# B&R Automation Studio project EFI (part 6)

### gAlrCore.mpalarmxcore - PC_any/mappServices/gAlrCore.mpalarmxcore
```
Element gAlrCore (Type=mpalarmxcore)
  mapp.AlarmX.Core.Configuration:
    [0]:
      Name = Dryer.Alarm.GenCritical
      Message = {$IAT/Dryer.Alarm.GenCritical}
      Code = 10001
      Severity = 1
      Behavior = PersistentAlarm
        Acknowledge = 0
        ReactionUntilAcknowledged = FALSE
        DataUpdate:
          Activation:
            TimeStamp = TRUE
            Snippets = TRUE
        Recording:
          ActiveToInactive = TRUE
          UnacknowledgedToAcknowledged = FALSE
          AcknowledgedToUnacknowledged = FALSE
    [1]:
      Name = Dryer.Alarm.GenStop
      Message = {$IAT/Dryer.Alarm.GenStop}
      Code = 10002
      Severity = 1
      Behavior = PersistentAlarm
        Acknowledge = 0
        ReactionUntilAcknowledged = FALSE
        DataUpdate:
          Activation:
            TimeStamp = TRUE
            Snippets = TRUE
        Recording:
          ActiveToInactive = TRUE
          UnacknowledgedToAcknowledged = FALSE
          AcknowledgedToUnacknowledged = FALSE
    [2]:
      Name = Dryer.Alarm.GenStopDrying
      Message = {$IAT/Dryer.Alarm.GenStopDrying}
      Code = 10003
      Severity = 1
      Behavior = PersistentAlarm
        Acknowledge = 0
        ReactionUntilAcknowledged = FALSE
        DataUpdate:
          Activation:
            TimeStamp = TRUE
            Snippets = TRUE
        Recording:
          ActiveToInactive = TRUE
          UnacknowledgedToAcknowledged = FALSE
          AcknowledgedToUnacknowledged = FALSE
    [3]:
      Name = Dryer.Alarm.FanBreakers
      Message = {$IAT/Dryer.Alarm.FanBreakers}
      Code = 10004
      Severity = 1
      Behavior = PersistentAlarm
        Acknowledge = 0
        ReactionUntilAcknowledged = FALSE
        DataUpdate:
          Activation:
            TimeStamp = TRUE
            Snippets = TRUE
        Recording:
          ActiveToInactive = TRUE
          UnacknowledgedToAcknowledged = FALSE
          AcknowledgedToUnacknowledged = FALSE
    [4]:
      Name = Dryer.Alarm.FansPsu
      Message = {$IAT/Dryer.Alarm.FansPsu}
      Code = 10005
      Severity = 1
      Behavior = PersistentAlarm
        Acknowledge = 0
        ReactionUntilAcknowledged = FALSE
        DataUpdate:
          Activation:
            TimeStamp = TRUE
            Snippets = TRUE
        Recording:
          ActiveToInactive = TRUE
          UnacknowledgedToAcknowledged = FALSE
          AcknowledgedToUnacknowledged = FALSE
    [5]:
      Name = Dryer.Alarm.MainPsu
      Message = {$IAT/Dryer.Alarm.MainPsu}
      Code = 10006
      Severity = 1
      Behavior = PersistentAlarm
        Acknowledge = 0
        ReactionUntilAcknowledged = FALSE
        DataUpdate:
          Activation:
            TimeStamp = TRUE
            Snippets = TRUE
        Recording:
          ActiveToInactive = TRUE
          UnacknowledgedToAcknowledged = FALSE
          AcknowledgedToUnacknowledged = FALSE
    [6]:
      Name = Dryer.Alarm.MountedMedia
      Message = {$IAT/Dryer.Alarm.MountedMedia}
      Code = 10007
      Severity = 1
      Behavior = PersistentAlarm
        Acknowledge = 0
        ReactionUntilAcknowledged = FALSE
        DataUpdate:
          Activation:
            TimeStamp = TRUE
            Snippets = TRUE
        Recording:
          ActiveToInactive = TRUE
          UnacknowledgedToAcknowledged = FALSE
          AcknowledgedToUnacknowledged = FALSE
    [7]:
      Name = Dryer.Alarm.EstopFront
      Message = {$IAT/Dryer.Alarm.EstopFront}
      Code = 10008
      Severity = 1
      Behavior = PersistentAlarm
        Acknowledge = 0
        ReactionUntilAcknowledged = FALSE
        DataUpdate:
          Activation:
            TimeStamp = TRUE
            Snippets = TRUE
        Recording:
          ActiveToInactive = TRUE
          UnacknowledgedToAcknowledged = FALSE
          AcknowledgedToUnacknowledged = FALSE
    [8]:
      Name = Dryer.Alarm.EstopRear
      Message = {$IAT/Dryer.Alarm.EstopRear}
      Code = 10009
      Severity = 1
      Behavior = PersistentAlarm
        Acknowledge = 0
        ReactionUntilAcknowledged = FALSE
        DataUpdate:
          Activation:
            TimeStamp = TRUE
            Snippets = TRUE
        Recording:
          ActiveToInactive = TRUE
          UnacknowledgedToAcknowledged = FALSE
          AcknowledgedToUnacknowledged = FALSE
    [9]:
      Name = Dryer.Alarm.EstopRemote
      Message = {$IAT/Dryer.Alarm.EstopRemote}
      Code = 10011
      Severity = 1
      Behavior = PersistentAlarm
        Acknowledge = 0
        ReactionUntilAcknowledged = FALSE
        DataUpdate:
          Activation:
            TimeStamp = TRUE
            Snippets = TRUE
        Recording:
          ActiveToInactive = TRUE
          UnacknowledgedToAcknowledged = FALSE
          AcknowledgedToUnacknowledged = FALSE
    [10]:
      Name = Dryer.Alarm.WrongPhysConfig
      Message = {$IAT/Dryer.Alarm.WrongPhysConfig}
      Code = 10012
      Severity = 1
      Behavior = PersistentAlarm
        Acknowledge = 0
        ReactionUntilAcknowledged = FALSE
        DataUpdate:
          Activation:
            TimeStamp = TRUE
            Snippets = TRUE
        Recording:
          ActiveToInactive = TRUE
          UnacknowledgedToAcknowledged = FALSE
          AcknowledgedToUnacknowledged = FALSE
    [11]:
      Name = Dryer.Alarm.OvertorqueBelt
      Message = {$IAT/Dryer.Alarm.OvertorqueBelt}
      Code = 10013
      Severity = 1
      Behavior = PersistentAlarm
        Acknowledge = 0
        ReactionUntilAcknowledged = FALSE
        DataUpdate:
          Activation:
            TimeStamp = TRUE
            Snippets = TRUE
        Recording:
          ActiveToInactive = TRUE
          UnacknowledgedToAcknowledged = FALSE
          AcknowledgedToUnacknowledged = FALSE
    [12]:
      Name = Dryer.Alarm.OverTempBeltFast
      Message = {$IAT/Dryer.Alarm.OverTempBeltFast}
      Code = 10014
      Severity = 1
      Behavior = PersistentAlarm
        Acknowledge = 0
        ReactionUntilAcknowledged = FALSE
        DataUpdate:
          Activation:
            TimeStamp = TRUE
            Snippets = TRUE
        Recording:
          ActiveToInactive = TRUE
          UnacknowledgedToAcknowledged = FALSE
          AcknowledgedToUnacknowledged = FALSE
    [13]:
      Name = Dryer.Alarm.OverTempBeltSlow
      Message = {$IAT/Dryer.Alarm.OverTempBeltSlow}
      Code = 10015
      Severity = 1
      Behavior = PersistentAlarm
        Acknowledge = 0
        ReactionUntilAcknowledged = FALSE
        DataUpdate:
          Activation:
            TimeStamp = TRUE
            Snippets = TRUE
        Recording:
          ActiveToInactive = TRUE
          UnacknowledgedToAcknowledged = FALSE
          AcknowledgedToUnacknowledged = FALSE
    [14]:
      Name = Dryer.Alarm.FansPsu80
      Message = {$IAT/Dryer.Alarm.FansPsu80}
      Code = 15001
      Severity = 2
      Behavior = PersistentAlarm
        Acknowledge = 0
        ReactionUntilAcknowledged = FALSE
        DataUpdate:
          Activation:
            TimeStamp = TRUE
            Snippets = TRUE
        Recording:
          ActiveToInactive = TRUE
          UnacknowledgedToAcknowledged = FALSE
          AcknowledgedToUnacknowledged = FALSE
    [15]:
      Name = Dryer.Warning.MountedMediaInside
      Message = {$IAT/Dryer.Warning.MountedMediaInside}
      Code = 15002
      Severity = 2
      Behavior = PersistentAlarm
        Acknowledge = 0
        ReactionUntilAcknowledged = FALSE
        DataUpdate:
          Activation:
            TimeStamp = TRUE
            Snippets = TRUE
        Recording:
          ActiveToInactive = TRUE
          UnacknowledgedToAcknowledged = FALSE
          AcknowledgedToUnacknowledged = FALSE
    [16]:
      Name = Dryer.Warning.BeltTempSensError
      Message = {$IAT/Dryer.Warning.BeltTempSensError}
      Code = 15003
      Severity = 2
      Behavior = PersistentAlarm
        Acknowledge = 0
        ReactionUntilAcknowledged = FALSE
        DataUpdate:
          Activation:
            TimeStamp = TRUE
            Snippets = TRUE
        Recording:
          ActiveToInactive = TRUE
          UnacknowledgedToAcknowledged = FALSE
          AcknowledgedToUnacknowledged = FALSE
    [17]:
      Name = Dryer.Warning.BoardInTempSensError
      Message = {$IAT/Dryer.Warning.BoardInTempSensError}
      Code = 15004
      Severity = 2
      Behavior = PersistentAlarm
        Acknowledge = 0
        ReactionUntilAcknowledged = FALSE
        DataUpdate:
          Activation:
            TimeStamp = TRUE
            Snippets = TRUE
        Recording:
          ActiveToInactive = TRUE
          UnacknowledgedToAcknowledged = FALSE
          AcknowledgedToUnacknowledged = FALSE
    [18]:
      Name = Dryer.Warning.BoardOutTempSensError
      Message = {$IAT/Dryer.Warning.BoardOutTempSensError}
      Code = 15005
      Severity = 2
      Behavior = PersistentAlarm
        Acknowledge = 0
        ReactionUntilAcknowledged = FALSE
        DataUpdate:
          Activation:
            TimeStamp = TRUE
            Snippets = TRUE
        Recording:
          ActiveToInactive = TRUE
          UnacknowledgedToAcknowledged = FALSE
          AcknowledgedToUnacknowledged = FALSE
    [19]:
      Name = Dryer.Warning.AirBlowerInTempSensError
      Message = {$IAT/Dryer.Warning.AirBlowerInTempSensError}
      Code = 15006
      Severity = 2
      Behavior = PersistentAlarm
        Acknowledge = 0
        ReactionUntilAcknowledged = FALSE
        DataUpdate:
          Activation:
            TimeStamp = TRUE
            Snippets = TRUE
        Recording:
          ActiveToInactive = TRUE
          UnacknowledgedToAcknowledged = FALSE
          AcknowledgedToUnacknowledged = FALSE
    [20]:
      Name = Dryer.Warning.AirBlowerOutTempSensError
      Message = {$IAT/Dryer.Warning.AirBlowerOutTempSensError}
      Code = 15007
      Severity = 2
      Behavior = PersistentAlarm
        Acknowledge = 0
        ReactionUntilAcknowledged = FALSE
        DataUpdate:
          Activation:
            TimeStamp = TRUE
            Snippets = TRUE
        Recording:
          ActiveToInactive = TRUE
          UnacknowledgedToAcknowledged = FALSE
          AcknowledgedToUnacknowledged = FALSE
    [21]:
      Name = Dryer.Warning.FrontDoorOpened
      Message = {$IAT/Dryer.Warning.FrontDoorOpened}
      Code = 15008
      Severity = 2
      Behavior = PersistentAlarm
        Acknowledge = 0
        ReactionUntilAcknowledged = FALSE
        DataUpdate:
          Activation:
            TimeStamp = TRUE
            Snippets = TRUE
        Recording:
          ActiveToInactive = TRUE
          UnacknowledgedToAcknowledged = FALSE
          AcknowledgedToUnacknowledged = FALSE
    [22]:
      Name = Dryer.Warning.RearDoorOpened
      Message = {$IAT/Dryer.Warning.RearDoorOpened}
      Code = 15009
      Severity = 2
      Behavior = PersistentAlarm
        Acknowledge = 0
        ReactionUntilAcknowledged = FALSE
        DataUpdate:
          Activation:
            TimeStamp = TRUE
            Snippets = TRUE
        Recording:
          ActiveToInactive = TRUE
          UnacknowledgedToAcknowledged = FALSE
          AcknowledgedToUnacknowledged = FALSE
    [23]:
      Name = Dryer.Warning.BentMedia
      Message = {$IAT/Dryer.Warning.BentMedia}
      Code = 15010
      Severity = 2
      Behavior = PersistentAlarm
        Acknowledge = 0
        ReactionUntilAcknowledged = FALSE
        DataUpdate:
          Activation:
            TimeStamp = TRUE
            Snippets = TRUE
        Recording:
          ActiveToInactive = TRUE
          UnacknowledgedToAcknowledged = FALSE
          AcknowledgedToUnacknowledged = FALSE
    [24]:
      Name = Dryer.Warning.NotMovementEnabled
      Message = {$IAT/Dryer.Warning.NotMovementEnabled}
      Code = 15011
      Severity = 2
      Behavior = PersistentAlarm
        Acknowledge = 0
        ReactionUntilAcknowledged = FALSE
        DataUpdate:
          Activation:
            TimeStamp = TRUE
            Snippets = TRUE
        Recording:
          ActiveToInactive = TRUE
          UnacknowledgedToAcknowledged = FALSE
          AcknowledgedToUnacknowledged = FALSE
    [25]:
      Name = Dryer.Warning.KeyMantenance
      Message = {$IAT/Dryer.Warning.KeyMantenance}
      Code = 15013
      Severity = 2
      Behavior = PersistentAlarm
        Acknowledge = 0
        ReactionUntilAcknowledged = FALSE
        DataUpdate:
          Activation:
            TimeStamp = TRUE
            Snippets = TRUE
        Recording:
          ActiveToInactive = TRUE
          UnacknowledgedToAcknowledged = FALSE
          AcknowledgedToUnacknowledged = FALSE
    [26]:
      Name = Dryer.Warning.JamLowCrash
      Message = {$IAT/Dryer.Warning.JamLowCrash}
      Code = 15014
      Severity = 2
      Behavior = PersistentAlarm
        Acknowledge = 0
        ReactionUntilAcknowledged = FALSE
        DataUpdate:
          Activation:
            TimeStamp = TRUE
            Snippets = TRUE
        Recording:
          ActiveToInactive = TRUE
          UnacknowledgedToAcknowledged = FALSE
          AcknowledgedToUnacknowledged = FALSE
    [27]:
      Name = Dryer.Alarm.BeltAnyDriveAlarm
      Message = {$IAT/Dryer.Alarm.BeltAnyDriveAlarm}
      Code = 30002
      Severity = 1
      Behavior = PersistentAlarm
        Acknowledge = 0
        ReactionUntilAcknowledged = FALSE
        DataUpdate:
          Activation:
            TimeStamp = TRUE
            Snippets = TRUE
        Recording:
          ActiveToInactive = TRUE
          UnacknowledgedToAcknowledged = FALSE
          AcknowledgedToUnacknowledged = FALSE
    [28]:
      Name = Dryer.Alarm.BeltAlrPowerBeltError
      Message = {$IAT/Dryer.Alarm.BeltAlrPowerBeltError}
      Code = 30003
      Severity = 1
      Behavior = PersistentAlarm
        Acknowledge = 0
        ReactionUntilAcknowledged = FALSE
        DataUpdate:
          Activation:
            TimeStamp = TRUE
            Snippets = TRUE
        Recording:
          ActiveToInactive = TRUE
          UnacknowledgedToAcknowledged = FALSE
          AcknowledgedToUnacknowledged = FALSE
    [29]:
      Name = Dryer.Alarm.BeltAlrComDrive
      Message = {$IAT/Dryer.Alarm.BeltAlrComDrive}
      Code = 30004
      Severity = 1
      Behavior = PersistentAlarm
        Acknowledge = 0
        ReactionUntilAcknowledged = FALSE
        DataUpdate:
          Activation:
            TimeStamp = TRUE
            Snippets = TRUE
        Recording:
          ActiveToInactive = TRUE
          UnacknowledgedToAcknowledged = FALSE
          AcknowledgedToUnacknowledged = FALSE
    [30]:
      Name = Dryer.Alarm.BeltAlrProtDrive
      Message = {$IAT/Dryer.Alarm.BeltAlrProtDrive}
      Code = 30005
      Severity = 1
      Behavior = PersistentAlarm
        Acknowledge = 0
        ReactionUntilAcknowledged = FALSE
        DataUpdate:
          Activation:
            TimeStamp = TRUE
            Snippets = TRUE
        Recording:
          ActiveToInactive = TRUE
          UnacknowledgedToAcknowledged = FALSE
          AcknowledgedToUnacknowledged = FALSE
    [31]:
      Name = Dryer.Alarm.BeltAlrOverTorque
      Message = {$IAT/Dryer.Alarm.BeltAlrOverTorque}
      Code = 30006
      Severity = 1
      Behavior = PersistentAlarm
        Acknowledge = 0
        ReactionUntilAcknowledged = FALSE
        DataUpdate:
          Activation:
            TimeStamp = TRUE
            Snippets = TRUE
        Recording:
          ActiveToInactive = TRUE
          UnacknowledgedToAcknowledged = FALSE
          AcknowledgedToUnacknowledged = FALSE
    [32]:
      Name = Dryer.Alarm.BeltBeltMotorTemp
      Message = {$IAT/Dryer.Alarm.BeltBeltMotorTemp}
      Code = 30007
      Severity = 1
      Behavior = PersistentAlarm
        Acknowledge = 0
        ReactionUntilAcknowledged = FALSE
        DataUpdate:
          Activation:
            TimeStamp = TRUE
            Snippets = TRUE
        Recording:
          ActiveToInactive = TRUE
          UnacknowledgedToAcknowledged = FALSE
          AcknowledgedToUnacknowledged = FALSE
    [33]:
      Name = Dryer.Alarm.BeltBeltDriverTemp
      Message = {$IAT/Dryer.Alarm.BeltBeltDriverTemp}
      Code = 30008
      Severity = 1
      Behavior = PersistentAlarm
        Acknowledge = 0
        ReactionUntilAcknowledged = FALSE
        DataUpdate:
          Activation:
            TimeStamp = TRUE
            Snippets = TRUE
        Recording:
          ActiveToInactive = TRUE
          UnacknowledgedToAcknowledged = FALSE
          AcknowledgedToUnacknowledged = FALSE
    [34]:
      Name = Dryer.Alarm.BeltNoPerimeter
      Message = {$IAT/Dryer.Alarm.BeltNoPerimeter}
      Code = 30009
      Severity = 2
      Behavior = PersistentAlarm
        Acknowledge = 0
        ReactionUntilAcknowledged = FALSE
        DataUpdate:
          Activation:
            TimeStamp = TRUE
            Snippets = TRUE
        Recording:
          ActiveToInactive = TRUE
          UnacknowledgedToAcknowledged = FALSE
          AcknowledgedToUnacknowledged = FALSE
    [35]:
      Name = Dryer.Alarm.BeltNoGearBox
      Message = {$IAT/Dryer.Alarm.BeltNoGearBox}
      Code = 30010
      Severity = 2
      Behavior = PersistentAlarm
        Acknowledge = 0
        ReactionUntilAcknowledged = FALSE
        DataUpdate:
          Activation:
            TimeStamp = TRUE
            Snippets = TRUE
        Recording:
          ActiveToInactive = TRUE
          UnacknowledgedToAcknowledged = FALSE
          AcknowledgedToUnacknowledged = FALSE
    [36]:
      Name = Dryer.Alarm.xWarningOvertoque
      Message = {$IAT/Dryer.Alarm.xWarningOvertoque}
      Code = 30102
      Severity = 2
      Behavior = PersistentAlarm
        Acknowledge = 0
        ReactionUntilAcknowledged = FALSE
        DataUpdate:
          Activation:
            TimeStamp = TRUE
            Snippets = TRUE
        Recording:
          ActiveToInactive = TRUE
          UnacknowledgedToAcknowledged = FALSE
          AcknowledgedToUnacknowledged = FALSE
    [37]:
      Name = Dryer.Alarm.SblockNotReferenced
      Message = {$IAT/Dryer.Alarm.SblockNotReferenced}
      Code = 40001
      Severity = 1
      Behavior = PersistentAlarm
        Acknowledge = 0
        ReactionUntilAcknowledged = FALSE
        DataUpdate:
          Activation:
            TimeStamp = TRUE
            Snippets = TRUE
        Recording:
          ActiveToInactive = TRUE
          UnacknowledgedToAcknowledged = FALSE
          AcknowledgedToUnacknowledged = FALSE
    [38]:
      Name = Dryer.Alarm.SblockNotCommsDrive
      Message = {$IAT/Dryer.Alarm.SblockNotCommsDrive}
      Code = 40002
      Severity = 1
      Behavior = PersistentAlarm
        Acknowledge = 0
        ReactionUntilAcknowledged = FALSE
        DataUpdate:
          Activation:
            TimeStamp = TRUE
            Snippets = TRUE
        Recording:
          ActiveToInactive = TRUE
          UnacknowledgedToAcknowledged = FALSE
          AcknowledgedToUnacknowledged = FALSE
    [39]:
      Name = Dryer.Alarm.SblockDriveBreaker
      Message = {$IAT/Dryer.Alarm.SblockDriveBreaker}
      Code = 40003
      Severity = 1
      Behavior = PersistentAlarm
        Acknowledge = 0
        ReactionUntilAcknowledged = FALSE
        DataUpdate:
          Activation:
            TimeStamp = TRUE
            Snippets = TRUE
        Recording:
          ActiveToInactive = TRUE
          UnacknowledgedToAcknowledged = FALSE
          AcknowledgedToUnacknowledged = FALSE
    [40]:
      Name = Dryer.Alarm.SblockHomeSensorError
      Message = {$IAT/Dryer.Alarm.SblockHomeSensorError}
      Code = 40004
      Severity = 1
      Behavior = PersistentAlarm
        Acknowledge = 0
        ReactionUntilAcknowledged = FALSE
        DataUpdate:
          Activation:
            TimeStamp = TRUE
            Snippets = TRUE
        Recording:
          ActiveToInactive = TRUE
          UnacknowledgedToAcknowledged = FALSE
          AcknowledgedToUnacknowledged = FALSE
    [41]:
      Name = Dryer.Alarm.SblockCheckHomeSensor
      Message = {$IAT/Dryer.Alarm.SblockCheckHomeSensor}
      Code = 40051
      Severity = 2
      Behavior = PersistentAlarm
        Acknowledge = 0
        ReactionUntilAcknowledged = FALSE
        DataUpdate:
          Activation:
            TimeStamp = TRUE
            Snippets = TRUE
        Recording:
          ActiveToInactive = TRUE
          UnacknowledgedToAcknowledged = FALSE
          AcknowledgedToUnacknowledged = FALSE
    [42]:
      Name = Dryer.Alarm.SblockMotorTemp
      Message = {$IAT/Dryer.Alarm.SblockMotorTemp}
      Code = 40052
      Severity = 2
      Behavior = PersistentAlarm
        Acknowledge = 0
        ReactionUntilAcknowledged = FALSE
        DataUpdate:
          Activation:
            TimeStamp = TRUE
            Snippets = TRUE
        Recording:
          ActiveToInactive = TRUE
          UnacknowledgedToAcknowledged = FALSE
          AcknowledgedToUnacknowledged = FALSE
    [43]:
      Name = Dryer.Alarm.SblockDriveTemp
      Message = {$IAT/Dryer.Alarm.SblockDriveTemp}
      Code = 40053
      Severity = 2
      Behavior = PersistentAlarm
        Acknowledge = 0
        ReactionUntilAcknowledged = FALSE
        DataUpdate:
          Activation:
            TimeStamp = TRUE
            Snippets = TRUE
        Recording:
          ActiveToInactive = TRUE
          UnacknowledgedToAcknowledged = FALSE
          AcknowledgedToUnacknowledged = FALSE
    [44]:
      Name = Dryer.Alarm.VaccSensor
      Message = {$IAT/Dryer.Alarm.VaccSensor}
      Code = 50001
      Severity = 1
      Behavior = PersistentAlarm
        Acknowledge = 0
        ReactionUntilAcknowledged = FALSE
        DataUpdate:
          Activation:
            TimeStamp = TRUE
            Snippets = TRUE
        Recording:
          ActiveToInactive = TRUE
          UnacknowledgedToAcknowledged = FALSE
          AcknowledgedToUnacknowledged = FALSE
    [45]:
      Name = Dryer.Alarm.VaccBlowerComsInput
      Message = {$IAT/Dryer.Alarm.VaccBlowerComsInput}
      Code = 50051
      Severity = 1
      Behavior = PersistentAlarm
        Acknowledge = 0
        ReactionUntilAcknowledged = FALSE
        DataUpdate:
          Activation:
            TimeStamp = TRUE
            Snippets = TRUE
        Recording:
          ActiveToInactive = TRUE
          UnacknowledgedToAcknowledged = FALSE
          AcknowledgedToUnacknowledged = FALSE
    [46]:
      Name = Dryer.Alarm.VaccBlowerComsOutput
      Message = {$IAT/Dryer.Alarm.VaccBlowerComsOutput}
      Code = 50052
      Severity = 1
      Behavior = PersistentAlarm
        Acknowledge = 0
        ReactionUntilAcknowledged = FALSE
        DataUpdate:
          Activation:
            TimeStamp = TRUE
            Snippets = TRUE
        Recording:
          ActiveToInactive = TRUE
          UnacknowledgedToAcknowledged = FALSE
          AcknowledgedToUnacknowledged = FALSE
    [47]:
      Name = Dryer.Alarm.VaccBlowerProtInput
      Message = {$IAT/Dryer.Alarm.VaccBlowerProtInput}
      Code = 50061
      Severity = 1
      Behavior = PersistentAlarm
        Acknowledge = 0
        ReactionUntilAcknowledged = FALSE
        DataUpdate:
          Activation:
            TimeStamp = TRUE
            Snippets = TRUE
        Recording:
          ActiveToInactive = TRUE
          UnacknowledgedToAcknowledged = FALSE
          AcknowledgedToUnacknowledged = FALSE
    [48]:
      Name = Dryer.Alarm.VaccBlowerProtOutput
      Message = {$IAT/Dryer.Alarm.VaccBlowerProtOutput}
      Code = 50062
      Severity = 1
      Behavior = PersistentAlarm
        Acknowledge = 0
        ReactionUntilAcknowledged = FALSE
        DataUpdate:
          Activation:
            TimeStamp = TRUE
            Snippets = TRUE
        Recording:
          ActiveToInactive = TRUE
          UnacknowledgedToAcknowledged = FALSE
          AcknowledgedToUnacknowledged = FALSE
    [49]:
      Name = Dryer.Alarm.VaccBlowerErrorInput
      Message = {$IAT/Dryer.Alarm.VaccBlowerErrorInput}
      Code = 50071
      Severity = 1
      Behavior = PersistentAlarm
        Acknowledge = 0
        ReactionUntilAcknowledged = FALSE
        DataUpdate:
          Activation:
            TimeStamp = TRUE
            Snippets = TRUE
        Recording:
          ActiveToInactive = TRUE
          UnacknowledgedToAcknowledged = FALSE
          AcknowledgedToUnacknowledged = FALSE
    [50]:
      Name = Dryer.Alarm.VaccBlowerErrorOutput
      Message = {$IAT/Dryer.Alarm.VaccBlowerErrorOutput}
      Code = 50072
      Severity = 1
      Behavior = PersistentAlarm
        Acknowledge = 0
        ReactionUntilAcknowledged = FALSE
        DataUpdate:
          Activation:
            TimeStamp = TRUE
            Snippets = TRUE
        Recording:
          ActiveToInactive = TRUE
          UnacknowledgedToAcknowledged = FALSE
          AcknowledgedToUnacknowledged = FALSE
    [51]:
      Name = Dryer.Alarm.VaccBlowerNotRunningInput
      Message = {$IAT/Dryer.Alarm.VaccBlowerNotRunningInput}
      Code = 50081
      Severity = 1
      Behavior = PersistentAlarm
        Acknowledge = 0
        ReactionUntilAcknowledged = FALSE
        DataUpdate:
          Activation:
            TimeStamp = TRUE
            Snippets = TRUE
        Recording:
          ActiveToInactive = TRUE
          UnacknowledgedToAcknowledged = FALSE
          AcknowledgedToUnacknowledged = FALSE
    [52]:
      Name = Dryer.Alarm.VaccBlowerNotRunningOutput
      Message = {$IAT/Dryer.Alarm.VaccBlowerNotRunningOutput}
      Code = 50082
      Severity = 1
      Behavior = PersistentAlarm
        Acknowledge = 0
        ReactionUntilAcknowledged = FALSE
        DataUpdate:
          Activation:
            TimeStamp = TRUE
            Snippets = TRUE
        Recording:
          ActiveToInactive = TRUE
          UnacknowledgedToAcknowledged = FALSE
          AcknowledgedToUnacknowledged = FALSE
    [53]:
      Name = Dryer.Alarm.NIRSafetyError
      Message = {$IAT/Dryer.Alarm.NIRSafetyError}
      Code = 60001
      Severity = 1
      Behavior = PersistentAlarm
        Acknowledge = 0
        ReactionUntilAcknowledged = FALSE
        DataUpdate:
          Activation:
            TimeStamp = TRUE
            Snippets = TRUE
        Recording:
          ActiveToInactive = TRUE
          UnacknowledgedToAcknowledged = FALSE
          AcknowledgedToUnacknowledged = FALSE
    [54]:
      Name = Dryer.Alarm.NIRFault
      Message = {$IAT/Dryer.Alarm.NIRFault}
      Code = 60002
      Severity = 1
      Behavior = PersistentAlarm
        Acknowledge = 0
        ReactionUntilAcknowledged = FALSE
        DataUpdate:
          Activation:
            TimeStamp = TRUE
            Snippets = TRUE
        Recording:
          ActiveToInactive = TRUE
          UnacknowledgedToAcknowledged = FALSE
          AcknowledgedToUnacknowledged = FALSE
    [55]:
      Name = Dryer.Alarm.NIRComsError
      Message = {$IAT/Dryer.Alarm.NIRComsError}
      Code = 60003
      Severity = 1
      Behavior = PersistentAlarm
        Acknowledge = 0
        ReactionUntilAcknowledged = FALSE
        DataUpdate:
          Activation:
            TimeStamp = TRUE
            Snippets = TRUE
        Recording:
          ActiveToInactive = TRUE
          UnacknowledgedToAcknowledged = FALSE
          AcknowledgedToUnacknowledged = FALSE
    [56]:
      Name = Dryer.Alarm.NIRInletHumiditySensError
      Message = {$IAT/Dryer.Alarm.NIRInletHumiditySensError}
      Code = 60021
      Severity = 2
      Behavior = PersistentAlarm
        Acknowledge = 0
        ReactionUntilAcknowledged = FALSE
        DataUpdate:
          Activation:
            TimeStamp = TRUE
            Snippets = TRUE
        Recording:
          ActiveToInactive = TRUE
          UnacknowledgedToAcknowledged = FALSE
          AcknowledgedToUnacknowledged = FALSE
    [57]:
      Name = Dryer.Alarm.NIRInletTempSensError
      Message = {$IAT/Dryer.Alarm.NIRInletTempSensError}
      Code = 60022
      Severity = 2
      Behavior = PersistentAlarm
        Acknowledge = 0
        ReactionUntilAcknowledged = FALSE
        DataUpdate:
          Activation:
            TimeStamp = TRUE
            Snippets = TRUE
        Recording:
          ActiveToInactive = TRUE
          UnacknowledgedToAcknowledged = FALSE
          AcknowledgedToUnacknowledged = FALSE
    [58]:
      Name = Dryer.Alarm.JamInputNIR1
      Message = {$IAT/Dryer.Alarm.JamInputNIR1}
      Code = 60051
      Severity = 1
      Behavior = PersistentAlarm
        Acknowledge = 0
        ReactionUntilAcknowledged = FALSE
        DataUpdate:
          Activation:
            TimeStamp = TRUE
            Snippets = TRUE
        Recording:
          ActiveToInactive = TRUE
          UnacknowledgedToAcknowledged = FALSE
          AcknowledgedToUnacknowledged = FALSE
    [59]:
      Name = Dryer.Alarm.JamOutputNIR1
      Message = {$IAT/Dryer.Alarm.JamOutputNIR1}
      Code = 60052
      Severity = 1
      Behavior = PersistentAlarm
        Acknowledge = 0
        ReactionUntilAcknowledged = FALSE
        DataUpdate:
          Activation:
            TimeStamp = TRUE
            Snippets = TRUE
        Recording:
          ActiveToInactive = TRUE
          UnacknowledgedToAcknowledged = FALSE
          AcknowledgedToUnacknowledged = FALSE
    [60]:
      Name = Dryer.Alarm.JamInputNIR2
      Message = {$IAT/Dryer.Alarm.JamInputNIR2}
      Code = 60061
      Severity = 1
      Behavior = PersistentAlarm
        Acknowledge = 0
        ReactionUntilAcknowledged = FALSE
        DataUpdate:
          Activation:
            TimeStamp = TRUE
            Snippets = TRUE
        Recording:
          ActiveToInactive = TRUE
          UnacknowledgedToAcknowledged = FALSE
          AcknowledgedToUnacknowledged = FALSE
    [61]:
      Name = Dryer.Alarm.JamOutputNIR2
      Message = {$IAT/Dryer.Alarm.JamOutputNIR2}
      Code = 60062
      Severity = 1
      Behavior = PersistentAlarm
        Acknowledge = 0
        ReactionUntilAcknowledged = FALSE
        DataUpdate:
          Activation:
            TimeStamp = TRUE
            Snippets = TRUE
        Recording:
          ActiveToInactive = TRUE
          UnacknowledgedToAcknowledged = FALSE
          AcknowledgedToUnacknowledged = FALSE
    [62]:
      Name = Dryer.Alarm.JamRearNIR1
      Message = {$IAT/Dryer.Alarm.JamRearNIR1}
      Code = 60071
      Severity = 1
      Behavior = PersistentAlarm
        Acknowledge = 0
        ReactionUntilAcknowledged = FALSE
        DataUpdate:
          Activation:
            TimeStamp = TRUE
            Snippets = TRUE
        Recording:
          ActiveToInactive = TRUE
          UnacknowledgedToAcknowledged = FALSE
          AcknowledgedToUnacknowledged = FALSE
    [63]:
      Name = Dryer.Alarm.JamRearNIR2
      Message = {$IAT/Dryer.Alarm.JamRearNIR2}
      Code = 60072
      Severity = 1
      Behavior = PersistentAlarm
        Acknowledge = 0
        ReactionUntilAcknowledged = FALSE
        DataUpdate:
          Activation:
            TimeStamp = TRUE
            Snippets = TRUE
        Recording:
          ActiveToInactive = TRUE
          UnacknowledgedToAcknowledged = FALSE
          AcknowledgedToUnacknowledged = FALSE
    [64]:
      Name = Dryer.Alarm.JamMechCrossNIR1
      Message = {$IAT/Dryer.Alarm.JamMechCrossNIR1}
      Code = 60081
      Severity = 1
      Behavior = PersistentAlarm
        Acknowledge = 0
        ReactionUntilAcknowledged = FALSE
        DataUpdate:
          Activation:
            TimeStamp = TRUE
            Snippets = TRUE
        Recording:
          ActiveToInactive = TRUE
          UnacknowledgedToAcknowledged = FALSE
          AcknowledgedToUnacknowledged = FALSE
    [65]:
      Name = Dryer.Alarm.JamMechCrossNIR2
      Message = {$IAT/Dryer.Alarm.JamMechCrossNIR2}
      Code = 60082
      Severity = 1
      Behavior = PersistentAlarm
        Acknowledge = 0
        ReactionUntilAcknowledged = FALSE
        DataUpdate:
          Activation:
            TimeStamp = TRUE
            Snippets = TRUE
        Recording:
          ActiveToInactive = TRUE
          UnacknowledgedToAcknowledged = FALSE
          AcknowledgedToUnacknowledged = FALSE
    [66]:
      Name = Dryer.Alarm.NIRSurfaceTemp1
      Message = {$IAT/Dryer.Alarm.NIRSurfaceTemp1}
      Code = 60101
      Severity = 2
      Behavior = PersistentAlarm
        Acknowledge = 0
        ReactionUntilAcknowledged = FALSE
        DataUpdate:
          Activation:
            TimeStamp = TRUE
            Snippets = TRUE
        Recording:
          ActiveToInactive = TRUE
          UnacknowledgedToAcknowledged = FALSE
          AcknowledgedToUnacknowledged = FALSE
    [67]:
      Name = Dryer.Alarm.NIRSurfaceTemp2
      Message = {$IAT/Dryer.Alarm.NIRSurfaceTemp2}
      Code = 60102
      Severity = 2
      Behavior = PersistentAlarm
        Acknowledge = 0
        ReactionUntilAcknowledged = FALSE
        DataUpdate:
          Activation:
            TimeStamp = TRUE
            Snippets = TRUE
        Recording:
          ActiveToInactive = TRUE
          UnacknowledgedToAcknowledged = FALSE
          AcknowledgedToUnacknowledged = FALSE
    [68]:
      Name = Dryer.Alarm.NIRSurfaceTempSensErr1
      Message = {$IAT/Dryer.Alarm.NIRSurfaceTempSensErr1}
      Code = 60111
      Severity = 2
      Behavior = PersistentAlarm
        Acknowledge = 0
        ReactionUntilAcknowledged = FALSE
        DataUpdate:
          Activation:
            TimeStamp = TRUE
            Snippets = TRUE
        Recording:
          ActiveToInactive = TRUE
          UnacknowledgedToAcknowledged = FALSE
          AcknowledgedToUnacknowledged = FALSE
    [69]:
      Name = Dryer.Alarm.NIRSurfaceTempSensErr2
      Message = {$IAT/Dryer.Alarm.NIRSurfaceTempSensErr2}
      Code = 60112
      Severity = 2
      Behavior = PersistentAlarm
        Acknowledge = 0
        ReactionUntilAcknowledged = FALSE
        DataUpdate:
          Activation:
            TimeStamp = TRUE
            Snippets = TRUE
        Recording:
          ActiveToInactive = TRUE
          UnacknowledgedToAcknowledged = FALSE
          AcknowledgedToUnacknowledged = FALSE
    [70]:
      Name = Dryer.Alarm.BlockedFan1Nir1
      Message = {$IAT/Dryer.Alarm.BlockedFan1Nir1}
      Code = 60201
      Severity = 2
      Behavior = PersistentAlarm
        Acknowledge = 0
        ReactionUntilAcknowledged = FALSE
        DataUpdate:
          Activation:
            TimeStamp = TRUE
            Snippets = TRUE
        Recording:
          ActiveToInactive = TRUE
          UnacknowledgedToAcknowledged = FALSE
          AcknowledgedToUnacknowledged = FALSE
    [71]:
      Name = Dryer.Alarm.BlockedFan2Nir1
      Message = {$IAT/Dryer.Alarm.BlockedFan2Nir1}
      Code = 60202
      Severity = 2
      Behavior = PersistentAlarm
        Acknowledge = 0
        ReactionUntilAcknowledged = FALSE
        DataUpdate:
          Activation:
            TimeStamp = TRUE
            Snippets = TRUE
        Recording:
          ActiveToInactive = TRUE
          UnacknowledgedToAcknowledged = FALSE
          AcknowledgedToUnacknowledged = FALSE
    [72]:
      Name = Dryer.Alarm.BlockedFan3Nir1
      Message = {$IAT/Dryer.Alarm.BlockedFan3Nir1}
      Code = 60203
      Severity = 2
      Behavior = PersistentAlarm
        Acknowledge = 0
        ReactionUntilAcknowledged = FALSE
        DataUpdate:
          Activation:
            TimeStamp = TRUE
            Snippets = TRUE
        Recording:
          ActiveToInactive = TRUE
          UnacknowledgedToAcknowledged = FALSE
          AcknowledgedToUnacknowledged = FALSE
    [73]:
      Name = Dryer.Alarm.BlockedFan4Nir1
      Message = {$IAT/Dryer.Alarm.BlockedFan4Nir1}
      Code = 60204
      Severity = 2
      Behavior = PersistentAlarm
        Acknowledge = 0
        ReactionUntilAcknowledged = FALSE
        DataUpdate:
          Activation:
            TimeStamp = TRUE
            Snippets = TRUE
        Recording:
          ActiveToInactive = TRUE
          UnacknowledgedToAcknowledged = FALSE
          AcknowledgedToUnacknowledged = FALSE
    [74]:
      Name = Dryer.Alarm.BlockedFan1Nir2
      Message = {$IAT/Dryer.Alarm.BlockedFan1Nir2}
      Code = 60211
      Severity = 2
      Behavior = PersistentAlarm
        Acknowledge = 0
        ReactionUntilAcknowledged = FALSE
        DataUpdate:
          Activation:
            TimeStamp = TRUE
            Snippets = TRUE
        Recording:
          ActiveToInactive = TRUE
          UnacknowledgedToAcknowledged = FALSE
          AcknowledgedToUnacknowledged = FALSE
    [75]:
      Name = Dryer.Alarm.BlockedFan2Nir2
      Message = {$IAT/Dryer.Alarm.BlockedFan2Nir2}
      Code = 60212
      Severity = 2
      Behavior = PersistentAlarm
        Acknowledge = 0
        ReactionUntilAcknowledged = FALSE
        DataUpdate:
          Activation:
            TimeStamp = TRUE
            Snippets = TRUE
        Recording:
          ActiveToInactive = TRUE
          UnacknowledgedToAcknowledged = FALSE
          AcknowledgedToUnacknowledged = FALSE
    [76]:
      Name = Dryer.Alarm.BlockedFan3Nir2
      Message = {$IAT/Dryer.Alarm.BlockedFan3Nir2}
      Code = 60213
      Severity = 2
      Behavior = PersistentAlarm
        Acknowledge = 0
        ReactionUntilAcknowledged = FALSE
        DataUpdate:
          Activation:
            TimeStamp = TRUE
            Snippets = TRUE
        Recording:
          ActiveToInactive = TRUE
          UnacknowledgedToAcknowledged = FALSE
          AcknowledgedToUnacknowledged = FALSE
    [77]:
      Name = Dryer.Alarm.BlockedFan4Nir2
      Message = {$IAT/Dryer.Alarm.BlockedFan4Nir2}
      Code = 60214
      Severity = 2
      Behavior = PersistentAlarm
        Acknowledge = 0
        ReactionUntilAcknowledged = FALSE
        DataUpdate:
          Activation:
            TimeStamp = TRUE
            Snippets = TRUE
        Recording:
          ActiveToInactive = TRUE
          UnacknowledgedToAcknowledged = FALSE
          AcknowledgedToUnacknowledged = FALSE
    [78]:
      Name = Dryer.Alarm.ArcLampComsError
      Message = {$IAT/Dryer.Alarm.ArcLampComsError}
      Code = 70001
      Severity = 1
      Behavior = PersistentAlarm
        Acknowledge = 0
        ReactionUntilAcknowledged = FALSE
        DataUpdate:
          Activation:
            TimeStamp = TRUE
            Snippets = TRUE
        Recording:
          ActiveToInactive = TRUE
          UnacknowledgedToAcknowledged = FALSE
          AcknowledgedToUnacknowledged = FALSE
    [79]:
      Name = Dryer.Alarm.ArcLampCredentialsError
      Message = {$IAT/Dryer.Alarm.ArcLampCredentialsError}
      Code = 70002
      Severity = 1
      Behavior = PersistentAlarm
        Acknowledge = 0
        ReactionUntilAcknowledged = FALSE
        DataUpdate:
          Activation:
            TimeStamp = TRUE
            Snippets = TRUE
        Recording:
          ActiveToInactive = TRUE
          UnacknowledgedToAcknowledged = FALSE
          AcknowledgedToUnacknowledged = FALSE
    [80]:
      Name = Dryer.Alarm.ArcLampInternalError
      Message = {$IAT/Dryer.Alarm.ArcLampInternalError}
      Code = 70003
      Severity = 1
      Behavior = PersistentAlarm
        Acknowledge = 0
        ReactionUntilAcknowledged = FALSE
        DataUpdate:
          Activation:
            TimeStamp = TRUE
            Snippets = TRUE
        Recording:
          ActiveToInactive = TRUE
          UnacknowledgedToAcknowledged = FALSE
          AcknowledgedToUnacknowledged = FALSE
    [81]:
      Name = Dryer.Alarm.ArcLampJam
      Message = {$IAT/Dryer.Alarm.ArcLampJam}
      Code = 70004
      Severity = 1
      Behavior = PersistentAlarm
        Acknowledge = 0
        ReactionUntilAcknowledged = FALSE
        DataUpdate:
          Activation:
            TimeStamp = TRUE
            Snippets = TRUE
        Recording:
          ActiveToInactive = TRUE
          UnacknowledgedToAcknowledged = FALSE
          AcknowledgedToUnacknowledged = FALSE
    [82]:
      Name = Dryer.Alarm.ArcLampAlarmLamp1
      Message = {$IAT/Dryer.Alarm.ArcLampAlarmLamp1}
      Code = 70051
      Severity = 1
      Behavior = PersistentAlarm
        Acknowledge = 0
        ReactionUntilAcknowledged = FALSE
        DataUpdate:
          Activation:
            TimeStamp = TRUE
            Snippets = TRUE
        Recording:
          ActiveToInactive = TRUE
          UnacknowledgedToAcknowledged = FALSE
          AcknowledgedToUnacknowledged = FALSE
    [83]:
      Name = Dryer.Alarm.ArcLampAlarmLamp2
      Message = {$IAT/Dryer.Alarm.ArcLampAlarmLamp2}
      Code = 70052
      Severity = 1
      Behavior = PersistentAlarm
        Acknowledge = 0
        ReactionUntilAcknowledged = FALSE
        DataUpdate:
          Activation:
            TimeStamp = TRUE
            Snippets = TRUE
        Recording:
          ActiveToInactive = TRUE
          UnacknowledgedToAcknowledged = FALSE
          AcknowledgedToUnacknowledged = FALSE
    [84]:
      Name = Dryer.Alarm.CheckMediaExit1
      Message = {$IAT/Dryer.Alarm.CheckMediaExit1}
      Code = 80001
      Severity = 1
      Behavior = PersistentAlarm
        Acknowledge = 0
        ReactionUntilAcknowledged = FALSE
        DataUpdate:
          Activation:
            TimeStamp = TRUE
            Snippets = TRUE
        Recording:
          ActiveToInactive = TRUE
          UnacknowledgedToAcknowledged = FALSE
          AcknowledgedToUnacknowledged = FALSE
    [85]:
      Name = Dryer.Alarm.CheckMediaExit2
      Message = {$IAT/Dryer.Alarm.CheckMediaExit2}
      Code = 80002
      Severity = 1
      Behavior = PersistentAlarm
        Acknowledge = 0
        ReactionUntilAcknowledged = FALSE
        DataUpdate:
          Activation:
            TimeStamp = TRUE
            Snippets = TRUE
        Recording:
          ActiveToInactive = TRUE
          UnacknowledgedToAcknowledged = FALSE
          AcknowledgedToUnacknowledged = FALSE
  mapp.AlarmX.Core.Categories:
    [0]:
      Name = Critical
      SourceProperty:
        Severity = 1
    [1]:
      Name = Warning
      SourceProperty:
        Severity = 2
    [2]:
      Name = Message
      SourceProperty:
        Severity = 3
```

### gAlrHist.mpalarmxhistory - PC_any/mappServices/gAlrHist.mpalarmxhistory
```
Element gAlrHist (Type=mpalarmxhistory)
  mapp.AlarmX.History:
    Memory:
      MemorySize = 600
```

## Configuration SimTests

CPU , AutomationRuntime K4.93, Build 4.1.2, Safety 0.0, Vc V4.73.2

### Task classes (Cpu.sw)
```
Cyclic#1 (cycle 4000 us, tolerance 0 us):
  mappHMI <- (binary)
Cyclic#2 (cycle 8000 us, tolerance 0 us):
  Initialize <- Printer.Config.Initialize.prg
  InitAxisCo <- ExtPack._Motion.AxisCtrl.AxisCtrl_v2.InitAxisControl.prg
  Belt <- ExtPack._Motion.AxisCtrl.AxisCtrl_v2.AxisCtrl.prg
  BK_A <- ExtPack._Motion.AxisCtrl.AxisCtrl_v2.AxisCtrl.prg
  BK_B <- ExtPack._Motion.AxisCtrl.AxisCtrl_v2.AxisCtrl.prg
  Stepper3L <- ExtPack._Motion.AxisCtrl.AxisCtrl_v2.AxisCtrl.prg
  Gear3L <- ExtPack._Motion.AxisCtrl.AxisCtrl_v2.AxisCtrl.prg
  NoCrash1 <- ExtPack._Motion.AxisCtrl.AxisCtrl_v2.AxisCtrl.prg
  NoCrash2 <- ExtPack._Motion.AxisCtrl.AxisCtrl_v2.AxisCtrl.prg
  InitInvert <- ExtPack._Motion.InverterCtrl.InverterCtrl_v1.InitInverterCtrl.prg
  Inverter1 <- ExtPack._Motion.InverterCtrl.InverterCtrl_v1.InverterCtrl.prg
  Inverter2 <- ExtPack._Motion.InverterCtrl.InverterCtrl_v1.InverterCtrl.prg
  Inverter3 <- ExtPack._Motion.InverterCtrl.InverterCtrl_v1.InverterCtrl.prg
  Inverter4 <- ExtPack._Motion.InverterCtrl.InverterCtrl_v1.InverterCtrl.prg
  InitIclaSi <- ExtPack._Motion.IclaCtrl.IclaSim.IclaSim_v1.InitIclaSim.prg
  IclaSim1 <- ExtPack._Motion.IclaCtrl.IclaSim.IclaSim_v1.IclaSim.prg
  IclaSim2 <- ExtPack._Motion.IclaCtrl.IclaSim.IclaSim_v1.IclaSim.prg
  IclanLas <- ExtPack._Motion.IclaCtrl.IclaSim.IclaSim_v1.IclaSim.prg
  IclaEhd1 <- ExtPack._Motion.IclaCtrl.IclaSim.IclaSim_v1.IclaSim.prg
  IclaEhd2 <- ExtPack._Motion.IclaCtrl.IclaSim.IclaSim_v1.IclaSim.prg
  IclaEhd3 <- ExtPack._Motion.IclaCtrl.IclaSim.IclaSim_v1.IclaSim.prg
  IclaEhd4 <- ExtPack._Motion.IclaCtrl.IclaSim.IclaSim_v1.IclaSim.prg
  SimMachFst <- Printer.Sim.SimMachine_Fast.prg
  Analog_Fas <- ExtPack._Media.AnalogThicknessCtrl.AnalogThicknessCtrl_v1.Analog_Fast.prg
  nSens_Fast <- ExtPack._Media.nSensorCtrl.nSensorCtrl_v2.nSensorCtrl_Fast.prg
  Thick_Fast <- ExtPack._Media.ThicknessCtrl.ThicknessCtrl_v2.ThicknessCtrl_Fast.prg
Cyclic#4 (cycle 32000 us, tolerance 32000 us):
  PhysInp <- Printer.PhysicalMapping.PhysicalMapInputs.prg
  BlockInp <- Printer.BlockSignalsManager.BlockInputsMapping.prg
  SimMachine <- Printer.Sim.SimMachine.prg
  ThickSim <- ExtPack._Media.ThicknessCtrl.ThicknessCtrlSim.ThicknessCtrlSim_v1.ThicknessCtrlSim.prg
  ThickPos <- ExtPack._Media.ThicknessCtrl.ThicknessCtrl_v2.ThicknessCtrl.prg  // Thickness array manager
  LineCtrl <- LineCtrl.LineCtrl.prg
  Mach_Fast <- Printer.MachineCtrl.MachineCtrl_Fast.prg
  BeltCtrl <- ExtPack._Transport.BeltCtrl.BeltCtrl_v1.BeltCtrl.prg
  InitBlockC <- ExtPack.BlockCtrl.BlockCtrl_v1.InitBlockCtrl.prg
  Block_BK1 <- ExtPack.BlockCtrl.BlockCtrl_v1.BlockCtrl.prg
  Block_BK2 <- ExtPack.BlockCtrl.BlockCtrl_v1.BlockCtrl.prg
  AnalogThic <- ExtPack._Media.AnalogThicknessCtrl.AnalogThicknessCtrl_v1.AnalogThickness.prg
  nSensorCtr <- ExtPack._Media.nSensorCtrl.nSensorCtrl_v2.nSensorCtrl.prg
  InitChille <- ExtPack._Extras.ChillerCtrl.ChillerCtrl_v2.InitChiller.prg
  Chiller1 <- ExtPack._Extras.ChillerCtrl.ChillerCtrl_v2.ChillerCtrl.prg
  Chiller2 <- ExtPack._Extras.ChillerCtrl.ChillerCtrl_v2.ChillerCtrl.prg
  InitTransV <- ExtPack._Transport.TransVacuumCtrl.TransVacuumCtrl_v1.InitTransVacuumCtrl.prg
  TransVac1 <- ExtPack._Transport.TransVacuumCtrl.TransVacuumCtrl_v1.TransVacuumCtrl.prg
  TransVac2 <- ExtPack._Transport.TransVacuumCtrl.TransVacuumCtrl_v1.TransVacuumCtrl.prg
  InitNCrash <- ExtPack._Transport.NonCrashCtrl.NonCrashCtrl_v1.InitNonCrashCtrl.prg
  NonCrash1 <- ExtPack._Transport.NonCrashCtrl.NonCrashCtrl_v1.NonCrashCtrl.prg
  InitCuring <- ExtPack._Cure.CuringLedCtrl.CuringLedCtrl_v1.InitCuringLedCtrl.prg
  CuringLed1 <- ExtPack._Cure.CuringLedCtrl.CuringLedCtrl_v1.CuringLedCtrl.prg
  CuringLed2 <- ExtPack._Cure.CuringLedCtrl.CuringLedCtrl_v1.CuringLedCtrl.prg
  CuringLed3 <- ExtPack._Cure.CuringLedCtrl.CuringLedCtrl_v1.CuringLedCtrl.prg
  BlockOut <- Printer.BlockSignalsManager.BlockOutputsMapping.prg
  PhysOut <- Printer.PhysicalMapping.PhysicalMapOutputs.prg
  InitTraySi <- ExtPack._Tools.TestBench.TraySim.TraySim_v1.InitTraySim.prg
  TraySim1 <- ExtPack._Tools.TestBench.TraySim.TraySim_v1.TraySim.prg
  TraySim2 <- ExtPack._Tools.TestBench.TraySim.TraySim_v1.TraySim.prg
  InitBlockS <- ExtPack.BlockCtrl.BlockSim.BlockSim_v1.InitBlockSim.prg
  BlockSim1 <- ExtPack.BlockCtrl.BlockSim.BlockSim_v1.BlockSim.prg
  BlockSim2 <- ExtPack.BlockCtrl.BlockSim.BlockSim_v1.BlockSim.prg
  EhdCtrl <- ExtPack._Transport.EdgeHoldDown.EdgeHoldDown_v1.EdgeHoldDown.prg
  InitPaired <- ExtPack._Transport.PairedIclaMotors.PairedIclaMotors_v1.InitPairedIclaMotors.prg
  PairedIcl1 <- ExtPack._Transport.PairedIclaMotors.PairedIclaMotors_v1.PairedIclaMotors.prg
  PairedIcl2 <- ExtPack._Transport.PairedIclaMotors.PairedIclaMotors_v1.PairedIclaMotors.prg
  InitChilSi <- ExtPack._Extras.ChillerCtrl.ChillerSim.ChillerSim_v1.InitChillerSim.prg
  ChillSim1 <- ExtPack._Extras.ChillerCtrl.ChillerSim.ChillerSim_v1.ChillerSim.prg
  ChillSim2 <- ExtPack._Extras.ChillerCtrl.ChillerSim.ChillerSim_v1.ChillerSim.prg
  InitTrSim <- ExtPack._Transport.TransVacuumCtrl.TransVacuumSim.TransVacuumSim_v1.InitTransVacuumSim.prg
  TrVacSim1 <- ExtPack._Transport.TransVacuumCtrl.TransVacuumSim.TransVacuumSim_v1.TransVacuumSim.prg
  TrVacSim2 <- ExtPack._Transport.TransVacuumCtrl.TransVacuumSim.TransVacuumSim_v1.TransVacuumSim.prg
  TrVacSim3 <- ExtPack._Transport.TransVacuumCtrl.TransVacuumSim.TransVacuumSim_v1.TransVacuumSim.prg
  TrVacSim4 <- ExtPack._Transport.TransVacuumCtrl.TransVacuumSim.TransVacuumSim_v1.TransVacuumSim.prg
  InitCurSim <- ExtPack._Cure.CuringLedCtrl.CuringLedSim.CuringLedSim_v1.InitCuringLedSim.prg
  CurinSim1 <- ExtPack._Cure.CuringLedCtrl.CuringLedSim.CuringLedSim_v1.CuringLedSim.prg
  CurinSim2 <- ExtPack._Cure.CuringLedCtrl.CuringLedSim.CuringLedSim_v1.CuringLedSim.prg
  CurinSim3 <- ExtPack._Cure.CuringLedCtrl.CuringLedSim.CuringLedSim_v1.CuringLedSim.prg
  FeederCtrl <- ExtPack._Ancillaries.FeederCtrl.FeederCtrl_v1.FeederCtrl.prg
  PrimerCtrl <- ExtPack._Ancillaries.PrimerCtrl.PrimerCtrl_v1.PrimerCtrl.prg
  SarmCtrl <- ExtPack._Ancillaries.SarmCtrl.SarmCtrl.SarmCtrl.prg
  OpvCtrl <- ExtPack._Ancillaries.OpvCtrl.OpvCtrl_v1.OpvCtrl.prg
  StackerCtr <- ExtPack._Ancillaries.StackerCtrl.StackerCtrl_v1.StackerCtrl.prg
  DryerCtrl <- ExtPack._Ancillaries.DryerCtrl.DryerCtrl_v1.DryerCtrl.prg
  FeederSim <- ExtPack._Ancillaries.FeederCtrl.FeederSim.FeederSim_v1.FeederSim.prg
  SarmSim <- ExtPack._Ancillaries.SarmCtrl.SarmSim.SarmSim_v1.SarmSim.prg
  DryerSim <- Dryer.DryerSimAnc.DryerSimAnc_v1.DryerSimAnc.prg
  PrimerSim <- ExtPack._Ancillaries.PrimerCtrl.PrimerSim.PrimerSim_v1.PrimerSim.prg
  OpvSim <- ExtPack._Ancillaries.OpvCtrl.OpvSim.OpvSim_v1.OpvSim.prg
  SafeCtlSim <- ExtPack._Extras.SafetyControllerCtrl.SafetyControllerSim.SafetyControllerSim_v1.SafetyControllerSim.prg
  StackerSim <- ExtPack._Ancillaries.StackerCtrl.StackerSim.StackerSim_v1.StackerSim.prg
  InitJamDet <- ExtPack._Transport.JamDetectCtrl.JamDetect_v1.InitJamDetect.prg
  JamDetect1 <- ExtPack._Transport.JamDetectCtrl.JamDetect_v1.JamDetect.prg
  JamDetect2 <- ExtPack._Transport.JamDetectCtrl.JamDetect_v1.JamDetect.prg
  JamDetect3 <- ExtPack._Transport.JamDetectCtrl.JamDetect_v1.JamDetect.prg
  JamDetect4 <- ExtPack._Transport.JamDetectCtrl.JamDetect_v1.JamDetect.prg
  InitJamDeS <- ExtPack._Transport.JamDetectCtrl.JamDetectSim.JamDetectSim_v1.InitJamDetectSim.prg
  JamDetctS1 <- ExtPack._Transport.JamDetectCtrl.JamDetectSim.JamDetectSim_v1.JamDetectSim.prg
  JamDetctS2 <- ExtPack._Transport.JamDetectCtrl.JamDetectSim.JamDetectSim_v1.JamDetectSim.prg
  JamDetctS3 <- ExtPack._Transport.JamDetectCtrl.JamDetectSim.JamDetectSim_v1.JamDetectSim.prg
  JamDetctS4 <- ExtPack._Transport.JamDetectCtrl.JamDetectSim.JamDetectSim_v1.JamDetectSim.prg
  nSensorSim <- ExtPack._Media.nSensorCtrl.nSensorSim.nSensorSim_v1.nSensorSim.prg
  EhdSim <- ExtPack._Transport.EdgeHoldDown.EdgeHoldDownSim.EdgeHoldDownSim_v1.EdgeHoldDownSim.prg
  IniPairSim <- ExtPack._Transport.PairedIclaMotors.PairedIclaMotorsSim.PairedIclaMotorsSim_v1.InitPairedIclaMotorsSim.prg
  PairSim <- ExtPack._Transport.PairedIclaMotors.PairedIclaMotorsSim.PairedIclaMotorsSim_v1.PairedIclaMotorsSim.prg
  PairSim2 <- ExtPack._Transport.PairedIclaMotors.PairedIclaMotorsSim.PairedIclaMotorsSim_v1.PairedIclaMotorsSim.prg
  InitNonCra <- ExtPack._Transport.NonCrashCtrl.NonCrashSim.NonCrashSim_v1.InitNonCrashSim.prg
  NonCrashS1 <- ExtPack._Transport.NonCrashCtrl.NonCrashSim.NonCrashSim_v1.NonCrashSim.prg
Cyclic#5 (cycle 80000 us, tolerance 80000 us):
  InksInputs <- Printer.InksSignals.InksInputs.prg
  InitInksSi <- ExtPack.InksCtrl.InksSim.InksSim_v1.InitInksSim.prg
  InksSim01 <- ExtPack.InksCtrl.InksSim.InksSim_v1.InksSim.prg
  InksSim02 <- ExtPack.InksCtrl.InksSim.InksSim_v1.InksSim.prg
  InksSim03 <- ExtPack.InksCtrl.InksSim.InksSim_v1.InksSim.prg
  InksSim04 <- ExtPack.InksCtrl.InksSim.InksSim_v1.InksSim.prg
  InksSim05 <- ExtPack.InksCtrl.InksSim.InksSim_v1.InksSim.prg
  InksSim06 <- ExtPack.InksCtrl.InksSim.InksSim_v1.InksSim.prg
  InksSim07 <- ExtPack.InksCtrl.InksSim.InksSim_v1.InksSim.prg
  InksSim08 <- ExtPack.InksCtrl.InksSim.InksSim_v1.InksSim.prg
  InitIndex <- ExtPack.InksCtrl.InksCtrl_v3.InitInksCtrl.prg
  Inks_01 <- ExtPack.InksCtrl.InksCtrl_v3.InksCtrl.prg
  Inks_02 <- ExtPack.InksCtrl.InksCtrl_v3.InksCtrl.prg
  Inks_03 <- ExtPack.InksCtrl.InksCtrl_v3.InksCtrl.prg
  Inks_04 <- ExtPack.InksCtrl.InksCtrl_v3.InksCtrl.prg
  Inks_05 <- ExtPack.InksCtrl.InksCtrl_v3.InksCtrl.prg
  Inks_06 <- ExtPack.InksCtrl.InksCtrl_v3.InksCtrl.prg
  Inks_07 <- ExtPack.InksCtrl.InksCtrl_v3.InksCtrl.prg
  Inks_08 <- ExtPack.InksCtrl.InksCtrl_v3.InksCtrl.prg
  InksOutput <- Printer.InksSignals.InksOutputs.prg  // Physical outputs inks
  SafetySamp <- AsSafetySolution.SafetySample.prg
  EventLogGe <- ExtPack._Tools.EventLog.EventLog_v1.EventLogGen.prg
  SavePerman <- Printer.Config.SavePermanent.prg
  SimUseReg <- ExtPack._Tools.SimUseRegister.SimUseRegister_1.SimUseRegister.prg
Cyclic#6 (cycle 88000 us, tolerance 88000 us):
  SafetyCont <- ExtPack._Extras.SafetyControllerCtrl.SafetyControllerCtrl_v1.SafetyControllerCtrl.prg
  InitPowerM <- ExtPack._Extras.PowerMeterCtrl.PowerMeterCtrl_v1.InitPowerMeterCtrl.prg
  PowerMete1 <- ExtPack._Extras.PowerMeterCtrl.PowerMeterCtrl_v1.PowerMeterCtrl.prg
  PowerMete2 <- ExtPack._Extras.PowerMeterCtrl.PowerMeterCtrl_v1.PowerMeterCtrl.prg
  Mach_Conf <- Printer.Config.MachineConfigurator.prg  // Printer configurator program
  Mach_Slow <- Printer.MachineCtrl.MachineCtrl_Slow.prg
  ThickReadE <- ExtPack._Media.ThicknessCtrl.ThicknessCtrl_v2.ThickReadEnergy.prg
  BeltClean <- ExtPack._Transport.BeltCleaning.BeltCleaning_v1.BeltCleaning.prg
  BCleanSim <- ExtPack._Transport.BeltCleaning.BeltCleaningSim.BeltCleaningSim.prg
Cyclic#7 (cycle 44000 us, tolerance 88000 us):
  PLC2Kernel <- Printer.Comms.PLC2Kernel.prg
  ServModbus <- ExtPack._Comms.ModbusComms.ModbusComms_v1.ServModbus.prg
  Kernel2PLC <- Printer.Comms.Kernel2PLC.prg  // Comns Kernel to PLC
Cyclic#8 (cycle 16000 us, tolerance 16000 us):
  FunctionsT <- UnitTest.Tests.FunctionsTests.prg
  PrePrepare <- UnitTest.Tests.PrePrepare.prg
  PrepMach <- UnitTest.Tests.PrepareMachine.prg  // Prepare Machine to work properly in Sim
  BeltTests <- UnitTest.Tests.BeltTests.prg
  ConsTests <- UnitTest.Tests.ConsentTests.prg
  CleaningTe <- UnitTest.Tests.CleaningTests.prg
  LineTests <- UnitTest.Tests.LineTests.prg
  TrVacuumTe <- UnitTest.Tests.TrVacuumTests.prg
  BlockTests <- UnitTest.Tests.BlockTests.prg
  Cube <- UnitTest.Tests.Cube.prg
DataObjects: Acp10sys
NcDataObjects: AcpErrTxt <- AxisTables.AcpErrTxt.dob, acp10etxen <- AxisTables.acp10etxen.dob, SM_a <- AxisTables.SM_a.dob, SM_i <- AxisTables.SM_i.dob, BeltP4_a <- AxisTables.BeltP4_a.dob, BeltP4_i <- AxisTables.BeltP4_i.dob, BK1_a <- AxisTables.BK1_a.dob, BK1_i <- AxisTables.BK1_i.dob, BK_sim_a <- AxisTables.BK_sim_a.dob, NonCrash_a <- AxisTables.NonCrash_a.dob, NonCrash_i <- AxisTables.NonCrash_i.dob
VcDataObjects: SimVis <- Printer.Sim.SimVisu.dob, Panel <- AsSafetySolution.Panel.dob
Binaries: TCData, udbdef, vcfntttf, vcfile, vcshared, vcpdvnc, vcgclass, arial, SimVis03, arialxsr, vccslider, vcdsint, SimVis01, vccbtn, vcdsloc, vcpfar00, vccovl, vcmgr, vcctext, vcalarm, vcbclass, vcrt, vccnum, arialbd, vccshape, vcpdsw, vcnet, SimVis02, vctcal, vcpkat, vccstr, vcclbox, vccdt, vccurl, vccline, vccbar, vcchtml, vcxml, vccalarm, vcctrend, vccbmp, vccgauge, Panel01, Panel03, Panel02, vccddbox, vccpopup, TCLang, mvLoader, OpcUaSrv, arsvcreg, Acp10map, acp10cfg, User, Role, TC, ashwac, sysconf, ashwd, arconfig, asfw, iomap, Visu02, Visu03, Visu01, Diagn02, Diagn03, Diagn01, vcchspot, OpcUaMap
Libraries: UnitTest, LibAssert1, EFIAssert, UtWs, UtMgr, AsCANopen, FBs, Functions, ConvertFun, runtime, brsystem, sys_lib, standard, AsSafety, FileIO, AsXml, astime, asstring, AsFifo, NcGlobal, AsBrStr, BRSE_MBT, BRSE_MB, MTBasics, MTTypes, MTFilter, AsIecCon, AsIOAcc, AsBrMath, AsEPL, ArEventLog, Acp10_MC, Acp10par, Acp10sim, Acp10sdc, DataObj, EvLogLib, ArProject, AxisFunc, dvframe, AsSem, IecCheck, ThickLib, ErrACS380, Acp10man, MpAlarmX, MpBase, MpCom, MpServer, powerlnk, arssl, vcresman, ashttp, astcp, asopcuac, asopcuas, asmath, aruser, ashw, asarcfg
```

### Hardware
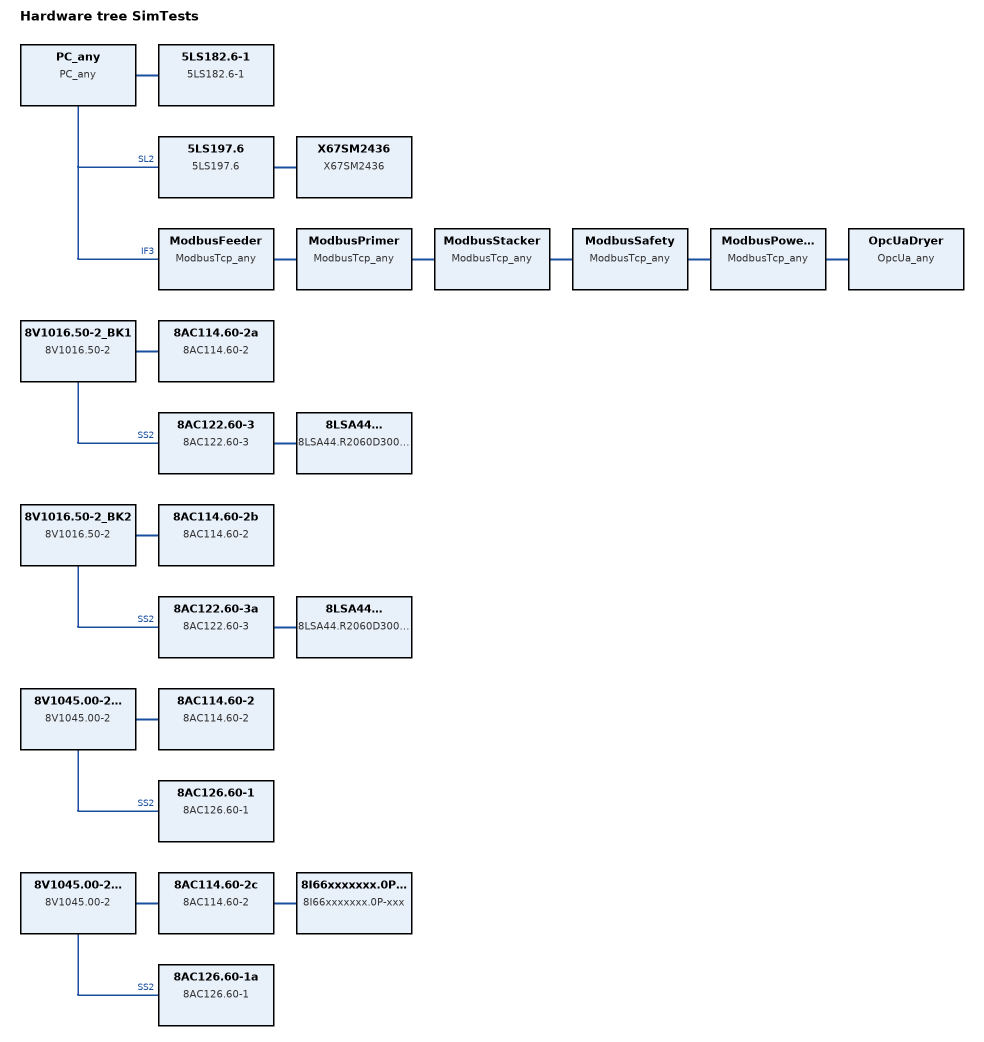
```
5LS182.6-1 : 5LS182.6-1 v1.5.0.0  [SL -> PC_any.SL1]
  Connector IF1:
    DNAConfiguration = manual
5LS197.6 : 5LS197.6 v1.1.0.0  [SL -> PC_any.SL2]
8AC114.60-2 : 8AC114.60-2 v1.0.0.8  [SS -> 8V1045.00-2_BELT.SS1; PLK1 -> 5LS182.6-1.IF1 [Cable Type=PowerlinkCable, Length=10, Version=1.0.0.3]; PLK2 -> 8AC114.60-2a.PLK1 [Cable Type=PowerlinkCable, Length=10, Version=1.0.0.3]]
8AC114.60-2a : 8AC114.60-2 v1.0.0.8  [SS -> 8V1016.50-2_BK1.SS1; PLK1 -> 8AC114.60-2.PLK2 [Cable Type=PowerlinkCable, Length=10, Version=1.0.0.3]; PLK2 -> 8AC114.60-2b.PLK1 [Cable Type=PowerlinkCable, Length=10, Version=1.0.0.3]]
8AC114.60-2b : 8AC114.60-2 v1.0.0.8  [SS -> 8V1016.50-2_BK2.SS1; PLK1 -> 8AC114.60-2a.PLK2 [Cable Type=PowerlinkCable, Length=10, Version=1.0.0.3]; PLK2 -> 8AC114.60-2c.PLK1 [Cable Type=PowerlinkCable, Length=10, Version=1.0.0.3]]
8AC114.60-2c : 8AC114.60-2 v1.0.0.8  [SS -> 8V1045.00-2_NCrash1.SS1; PLK1 -> 8AC114.60-2b.PLK2 [Cable Type=PowerlinkCable, Length=10, Version=1.0.0.3]; PLK2 -> 8I66xxxxxxx.0P-xxx1.PLK1 [Cable Type=PowerlinkCable, Length=10, Version=1.0.0.3]]
8AC122.60-3 : 8AC122.60-3 v2.2.0.0  [SS -> 8V1016.50-2_BK1.SS2]
8AC122.60-3a : 8AC122.60-3 v2.2.0.0  [SS -> 8V1016.50-2_BK2.SS2]
8AC126.60-1 : 8AC126.60-1 v2.2.0.0  [SS -> 8V1045.00-2_BELT.SS2]
8AC126.60-1a : 8AC126.60-1 v2.2.0.0  [SS -> 8V1045.00-2_NCrash1.SS2]
8I66xxxxxxx.0P-xxx1 : 8I66xxxxxxx.0P-xxx v2.5.1.0  [PLK1 -> 8AC114.60-2c.PLK2 [Cable Type=PowerlinkCable, Length=10, Version=1.0.0.3]]
  FunctionModel = Standard
  Supervision = off
  UnitOfSetpoint = Rpm
  IOM_AIDP1 = LFT
  IOM_AIDP2 = LCR
  IOM_AIDP3 = OTRN
  IOM_AIDP4 = IL1R
  IOM_AIDP5 = AI1R
  IOM_AIDP6 = AI2R
  IOM_AIDP7 = AI3R
  IOM_AIDP8 = OL1I
  IOM_AIDP9 = AO1I
  IOM_R1ctrl = mapped
  IOM_R2ctrl = mapped
  IOM_LO1ctrl = mapped
  IOM_AO1ctrl = mapped
  Sel_AO1T = 0A
  Sel_NameplateMask = MANU
  Cfg_NSP = 1400
  Cfg_UNS = 230
  Cfg_NCR = 19
  Cfg_COS = 71
  Cfg_NPR = 37
8LSA44.R2060D300-3 : 8LSA44.R2060D300-3 v2.2.0.0  [EC -> 8AC122.60-3.EC; MT -> 8V1016.50-2_BK1.MT1]
8LSA44.R2060D300-3a : 8LSA44.R2060D300-3 v2.2.0.0  [EC -> 8AC122.60-3a.EC; MT -> 8V1016.50-2_BK2.MT1]
8V1016.50-2_BK1 : 8V1016.50-2 v2.2.0.0
  MotionTP = Acp10Arnc0
8V1016.50-2_BK2 : 8V1016.50-2 v2.2.0.0
  MotionTP = Acp10Arnc0
8V1045.00-2_BELT : 8V1045.00-2 v2.2.0.0
  MotionTP = Acp10Arnc0
8V1045.00-2_NCrash1 : 8V1045.00-2 v2.2.0.0
  MotionTP = Acp10Arnc0
ModbusFeeder : ModbusTcp_any v1.1.0.0 (Disabled=true)  [ETH1 -> PC_any.IF3 [Cable Type=PowerlinkCable, Length=10, Version=1.0.0.3]; ETH2 -> ModbusPrimer.ETH1 [Cable Type=PowerlinkCable, Length=10, Version=1.0.0.3]]
  Connector ETH2 (Disabled=true)
  IpAddress = 192.168.125.175
  UnitId = 1
  Cb_1
  Cb_1_FunCode = 4
  Cb_1_NumItems = 25
  Cb_1_C_1
  Cb_1_C_1_Name = readFeederBk1_1
  Cb_1_C_1_Datatype = 6
  Cb_1_C_2
  Cb_1_C_2_Name = readFeederBk1_2
  Cb_1_C_2_Datatype = 6
  Cb_1_C_3
  Cb_1_C_3_Name = readFeederBk1_3
  Cb_1_C_3_Datatype = 6
  Cb_1_C_4
  Cb_1_C_4_Name = readFeederBk1_4
  Cb_1_C_4_Datatype = 6
  Cb_1_C_5
  Cb_1_C_5_Name = readFeederBk1_5
  Cb_1_C_5_Datatype = 6
  Cb_1_C_6
  Cb_1_C_6_Name = readFeederBk1_6
  Cb_1_C_6_Datatype = 6
  Cb_1_C_7
  Cb_1_C_7_Name = readFeederBk1_7
  Cb_1_C_7_Datatype = 6
  Cb_1_C_8
  Cb_1_C_8_Name = readFeederBk1_8
  Cb_1_C_8_Datatype = 6
  Cb_1_C_9
  Cb_1_C_9_Name = readFeederBk1_9
  Cb_1_C_9_Datatype = 6
  Cb_1_C_10
  Cb_1_C_10_Name = readFeederBk1_10
  Cb_1_C_10_Datatype = 6
  Cb_1_C_11
  Cb_1_C_11_Name = readFeederBk1_11
  Cb_1_C_11_Datatype = 6
  Cb_1_C_12
  Cb_1_C_12_Name = readFeederBk1_12
  Cb_1_C_12_Datatype = 6
  Cb_1_C_13
  Cb_1_C_13_Name = readFeederBk1_13
  Cb_1_C_13_Datatype = 6
  Cb_1_C_14
  Cb_1_C_14_Name = readFeederBk1_14
  Cb_1_C_14_Datatype = 6
  Cb_1_C_15
  Cb_1_C_15_Name = readFeederBk1_15
  Cb_1_C_15_Datatype = 6
  Cb_1_C_16
  Cb_1_C_16_Name = readFeederBk1_16
  Cb_1_C_16_Datatype = 6
  Cb_1_C_17
  Cb_1_C_17_Name = readFeederBk1_17
  Cb_1_C_17_Datatype = 6
  Cb_1_C_18
  Cb_1_C_18_Name = readFeederBk1_18
  Cb_1_C_18_Datatype = 6
  Cb_1_C_19
  Cb_1_C_19_Name = readFeederBk1_19
  Cb_1_C_19_Datatype = 6
  Cb_1_C_20
  Cb_1_C_20_Name = readFeederBk1_20
  Cb_1_C_20_Datatype = 6
  Cb_1_C_21
  Cb_1_C_21_Name = readFeederBk1_21
  Cb_1_C_21_Datatype = 6
  Cb_1_C_22
  Cb_1_C_22_Name = readFeederBk1_22
  Cb_1_C_22_Datatype = 6
  Cb_1_C_23
  Cb_1_C_23_Name = readFeederBk1_23
  Cb_1_C_23_Datatype = 6
  Cb_1_C_24
  Cb_1_C_24_Name = readFeederBk1_24
  Cb_1_C_24_Datatype = 6
  Cb_1_C_25
  Cb_1_C_25_Name = readFeederBk1_25
  Cb_1_C_25_Datatype = 6
  Cb_2
  Cb_2_FunCode = 16
  Cb_2_NumItemsExt = 25
  Cb_2_C_1
  Cb_2_C_1_Name = writeFeederBk2_1
  Cb_2_C_1_Datatype = 6
  Cb_2_C_1_Dir = 1
  Cb_2_C_2
  Cb_2_C_2_Name = writeFeederBk2_2
  Cb_2_C_2_Datatype = 6
  Cb_2_C_2_Dir = 1
  Cb_2_C_3
  Cb_2_C_3_Name = writeFeederBk2_3
  Cb_2_C_3_Datatype = 6
  Cb_2_C_3_Dir = 1
  Cb_2_C_4
  Cb_2_C_4_Name = writeFeederBk2_4
  Cb_2_C_4_Datatype = 6
  Cb_2_C_4_Dir = 1
  Cb_2_C_5
  Cb_2_C_5_Name = writeFeederBk2_5
  Cb_2_C_5_Datatype = 6
  Cb_2_C_5_Dir = 1
  Cb_2_C_6
  Cb_2_C_6_Name = writeFeederBk2_6
  Cb_2_C_6_Datatype = 6
  Cb_2_C_6_Dir = 1
  Cb_2_C_7
  Cb_2_C_7_Name = writeFeederBk2_7
  Cb_2_C_7_Datatype = 6
  Cb_2_C_7_Dir = 1
  Cb_2_C_8
  Cb_2_C_8_Name = writeFeederBk2_8
  Cb_2_C_8_Datatype = 6
  Cb_2_C_8_Dir = 1
  Cb_2_C_9
  Cb_2_C_9_Name = writeFeederBk2_9
  Cb_2_C_9_Datatype = 6
  Cb_2_C_9_Dir = 1
  Cb_2_C_10
  Cb_2_C_10_Name = writeFeederBk2_10
  Cb_2_C_10_Datatype = 6
  Cb_2_C_10_Dir = 1
  Cb_2_C_11
  Cb_2_C_11_Name = writeFeederBk2_11
  Cb_2_C_11_Datatype = 6
  Cb_2_C_11_Dir = 1
  Cb_2_C_12
  Cb_2_C_12_Name = writeFeederBk2_12
  Cb_2_C_12_Datatype = 6
  Cb_2_C_12_Dir = 1
  Cb_2_C_13
  Cb_2_C_13_Name = writeFeederBk2_13
  Cb_2_C_13_Datatype = 6
  Cb_2_C_13_Dir = 1
  Cb_2_C_14
  Cb_2_C_14_Name = writeFeederBk2_14
  Cb_2_C_14_Datatype = 6
  Cb_2_C_14_Dir = 1
  Cb_2_C_15
  Cb_2_C_15_Name = writeFeederBk2_15
  Cb_2_C_15_Datatype = 6
  Cb_2_C_15_Dir = 1
  Cb_2_C_16
  Cb_2_C_16_Name = writeFeederBk2_16
  Cb_2_C_16_Datatype = 6
  Cb_2_C_16_Dir = 1
  Cb_2_C_17
  Cb_2_C_17_Name = writeFeederBk2_17
  Cb_2_C_17_Datatype = 6
  Cb_2_C_17_Dir = 1
  Cb_2_C_18
  Cb_2_C_18_Name = writeFeederBk2_18
  Cb_2_C_18_Datatype = 6
  Cb_2_C_18_Dir = 1
  Cb_2_C_19
  Cb_2_C_19_Name = writeFeederBk2_19
  Cb_2_C_19_Datatype = 6
  Cb_2_C_19_Dir = 1
  Cb_2_C_20
  Cb_2_C_20_Name = writeFeederBk2_20
  Cb_2_C_20_Datatype = 6
  Cb_2_C_20_Dir = 1
  Cb_2_C_21
  Cb_2_C_21_Name = writeFeederBk2_21
  Cb_2_C_21_Datatype = 6
  Cb_2_C_21_Dir = 1
  Cb_2_C_22
  Cb_2_C_22_Name = writeFeederBk2_22
  Cb_2_C_22_Datatype = 6
  Cb_2_C_22_Dir = 1
  Cb_2_C_23
  Cb_2_C_23_Name = writeFeederBk2_23
  Cb_2_C_23_Datatype = 6
  Cb_2_C_23_Dir = 1
  Cb_2_C_24
  Cb_2_C_24_Name = writeFeederBk2_24
  Cb_2_C_24_Datatype = 6
  Cb_2_C_24_Dir = 1
  Cb_2_C_25
  Cb_2_C_25_Name = writeFeederBk2_25
  Cb_2_C_25_Datatype = 6
  Cb_2_C_25_Dir = 1
ModbusPowerMeter : ModbusTcp_any v1.1.0.0 (Disabled=true)  [ETH1 -> ModbusSafety.ETH2 [Cable Type=PowerlinkCable, Length=10, Version=1.0.0.3]; ETH2 -> OpcUaDryer.ETH1 [Cable Type=PowerlinkCable, Length=10, Version=1.0.0.3]]
  Connector ETH2 (Disabled=true)
  IpAddress = 192.168.125.210
  Cb_1
  Cb_1_FunCode = 3
  Cb_1_Addr = 12000
  Cb_1_NumItems = 0
  Cb_1_C_1
  Cb_1_C_1_Name = readPowerMeterBk1_1
  Cb_1_C_1_Datatype = 6
  Cb_1_C_2
  Cb_1_C_2_Name = readPowerMeterBk1_2
  Cb_1_C_2_Datatype = 6
  Cb_1_C_3
  Cb_1_C_3_Name = readPowerMeterBk1_3
  Cb_1_C_3_Datatype = 6
  Cb_1_C_4
  Cb_1_C_4_Name = readPowerMeterBk1_4
  Cb_1_C_4_Datatype = 6
  Cb_1_C_5
  Cb_1_C_5_Name = readPowerMeterBk1_5
  Cb_1_C_5_Datatype = 6
  Cb_1_C_6
  Cb_1_C_6_Name = readPowerMeterBk1_6
  Cb_1_C_6_Datatype = 6
  Cb_2
  Cb_2_FunCode = 3
  Cb_2_Addr = 12016
  Cb_2_NumItems = 0
  Cb_2_C_1
  Cb_2_C_1_Name = readPowerMeterBk2_1
  Cb_2_C_1_Datatype = 6
  Cb_2_C_2
  Cb_2_C_2_Name = readPowerMeterBk2_2
  Cb_2_C_2_Datatype = 6
  Cb_2_C_3
  Cb_2_C_3_Name = readPowerMeterBk2_3
  Cb_2_C_3_Datatype = 6
  Cb_2_C_4
  Cb_2_C_4_Name = readPowerMeterBk2_4
  Cb_2_C_4_Datatype = 6
  Cb_2_C_5
  Cb_2_C_5_Name = readPowerMeterBk2_5
  Cb_2_C_5_Datatype = 6
  Cb_2_C_6
  Cb_2_C_6_Name = readPowerMeterBk2_6
  Cb_2_C_6_Datatype = 6
  Cb_2_C_7
  Cb_2_C_7_Name = readPowerMeterBk2_7
  Cb_2_C_7_Datatype = 6
  Cb_2_C_8
  Cb_2_C_8_Name = readPowerMeterBk2_8
  Cb_2_C_8_Datatype = 6
  Cb_2_C_9
  Cb_2_C_9_Name = readPowerMeterBk2_9
  Cb_2_C_9_Datatype = 6
  Cb_2_C_10
  Cb_2_C_10_Name = readPowerMeterBk2_10
  Cb_2_C_10_Datatype = 6
  Cb_2_C_11
  Cb_2_C_11_Name = readPowerMeterBk2_11
  Cb_2_C_11_Datatype = 6
  Cb_2_C_12
  Cb_2_C_12_Name = readPowerMeterBk2_12
  Cb_2_C_12_Datatype = 6
  Cb_2_C_13
  Cb_2_C_13_Name = readPowerMeterBk2_13
  Cb_2_C_13_Datatype = 6
  Cb_2_C_14
  Cb_2_C_14_Name = readPowerMeterBk2_14
  Cb_2_C_14_Datatype = 6
  Cb_2_C_15
  Cb_2_C_15_Name = readPowerMeterBk2_15
  Cb_2_C_15_Datatype = 6
  Cb_2_C_16
  Cb_2_C_16_Name = readPowerMeterBk2_16
  Cb_2_C_16_Datatype = 6
  Cb_2_C_17
  Cb_2_C_17_Name = readPowerMeterBk2_17
  Cb_2_C_17_Datatype = 6
  Cb_2_C_18
  Cb_2_C_18_Name = readPowerMeterBk2_18
  Cb_2_C_18_Datatype = 6
  Cb_2_C_19
  Cb_2_C_19_Name = readPowerMeterBk2_19
  Cb_2_C_19_Datatype = 6
  Cb_2_C_20
  Cb_2_C_20_Name = readPowerMeterBk2_20
  Cb_2_C_20_Datatype = 6
  Cb_2_C_21
  Cb_2_C_21_Name = readPowerMeterBk2_21
  Cb_2_C_21_Datatype = 6
  Cb_2_C_22
  Cb_2_C_22_Name = readPowerMeterBk2_22
  Cb_2_C_22_Datatype = 6
  Cb_2_C_23
  Cb_2_C_23_Name = readPowerMeterBk2_23
  Cb_2_C_23_Datatype = 6
  Cb_2_C_24
  Cb_2_C_24_Name = readPowerMeterBk2_24
  Cb_2_C_24_Datatype = 6
  Cb_2_C_25
  Cb_2_C_25_Name = readPowerMeterBk2_25
  Cb_2_C_25_Datatype = 6
  Cb_2_C_26
  Cb_2_C_26_Name = readPowerMeterBk2_26
  Cb_2_C_26_Datatype = 6
  Cb_2_C_27
  Cb_2_C_27_Name = readPowerMeterBk2_27
  Cb_2_C_27_Datatype = 6
  Cb_2_C_28
  Cb_2_C_28_Name = readPowerMeterBk2_28
  Cb_2_C_28_Datatype = 6
  Cb_2_C_29
  Cb_2_C_29_Name = readPowerMeterBk2_29
  Cb_2_C_29_Datatype = 6
  Cb_2_C_30
  Cb_2_C_30_Name = readPowerMeterBk2_30
  Cb_2_C_30_Datatype = 6
  Cb_2_C_31
  Cb_2_C_31_Name = readPowerMeterBk2_31
  Cb_2_C_31_Datatype = 6
  Cb_2_C_32
  Cb_2_C_32_Name = readPowerMeterBk2_32
  Cb_2_C_32_Datatype = 6
  Cb_2_C_33
  Cb_2_C_33_Name = readPowerMeterBk2_33
  Cb_2_C_33_Datatype = 6
  Cb_2_C_34
  Cb_2_C_34_Name = readPowerMeterBk2_34
  Cb_2_C_34_Datatype = 6
  Cb_2_C_35
  Cb_2_C_35_Name = readPowerMeterBk2_35
  Cb_2_C_35_Datatype = 6
  Cb_3
  Cb_3_FunCode = 3
  Cb_3_Addr = 12104
  Cb_3_NumItems = 0
  Cb_3_C_1
  Cb_3_C_1_Name = readPowerMeterBk3_1
  Cb_3_C_1_Datatype = 6
  Cb_3_C_2
  Cb_3_C_2_Name = readPowerMeterBk3_2
  Cb_3_C_2_Datatype = 6
  Cb_3_C_3
  Cb_3_C_3_Name = readPowerMeterBk3_3
  Cb_3_C_3_Datatype = 6
  Cb_3_C_4
  Cb_3_C_4_Name = readPowerMeterBk3_4
  Cb_3_C_4_Datatype = 6
  Cb_3_C_5
  Cb_3_C_5_Name = readPowerMeterBk3_5
  Cb_3_C_5_Datatype = 6
  Cb_3_C_6
  Cb_3_C_6_Name = readPowerMeterBk3_6
  Cb_3_C_6_Datatype = 6
  Cb_3_C_7
  Cb_3_C_7_Name = readPowerMeterBk3_7
  Cb_3_C_7_Datatype = 6
  Cb_3_C_8
  Cb_3_C_8_Name = readPowerMeterBk3_8
  Cb_3_C_8_Datatype = 6
  Cb_3_C_9
  Cb_3_C_9_Name = readPowerMeterBk3_9
  Cb_3_C_9_Datatype = 6
  Cb_3_C_10
  Cb_3_C_10_Name = readPowerMeterBk3_10
  Cb_3_C_10_Datatype = 6
ModbusPrimer : ModbusTcp_any v1.1.0.0 (Disabled=true)  [ETH1 -> ModbusFeeder.ETH2 [Cable Type=PowerlinkCable, Length=10, Version=1.0.0.3]; ETH2 -> ModbusStacker.ETH1 [Cable Type=PowerlinkCable, Length=10, Version=1.0.0.3]]
  Connector ETH2 (Disabled=true)
  IpAddress = 192.168.125.130
  UnitId = 1
  Cb_1
  Cb_1_FunCode = 4
  Cb_1_NumItems = 25
  Cb_1_C_1
  Cb_1_C_1_Name = readCoaterBk1_1
  Cb_1_C_1_Datatype = 6
  Cb_1_C_2
  Cb_1_C_2_Name = readCoaterBk1_2
  Cb_1_C_2_Datatype = 6
  Cb_1_C_3
  Cb_1_C_3_Name = readCoaterBk1_3
  Cb_1_C_3_Datatype = 6
  Cb_1_C_4
  Cb_1_C_4_Name = readCoaterBk1_4
  Cb_1_C_4_Datatype = 6
  Cb_1_C_5
  Cb_1_C_5_Name = readCoaterBk1_5
  Cb_1_C_5_Datatype = 6
  Cb_1_C_6
  Cb_1_C_6_Name = readCoaterBk1_6
  Cb_1_C_6_Datatype = 6
  Cb_1_C_7
  Cb_1_C_7_Name = readCoaterBk1_7
  Cb_1_C_7_Datatype = 6
  Cb_1_C_8
  Cb_1_C_8_Name = readCoaterBk1_8
  Cb_1_C_8_Datatype = 6
  Cb_1_C_9
  Cb_1_C_9_Name = readCoaterBk1_9
  Cb_1_C_9_Datatype = 6
  Cb_1_C_10
  Cb_1_C_10_Name = readCoaterBk1_10
  Cb_1_C_10_Datatype = 6
  Cb_1_C_11
  Cb_1_C_11_Name = readCoaterBk1_11
  Cb_1_C_11_Datatype = 6
  Cb_1_C_12
  Cb_1_C_12_Name = readCoaterBk1_12
  Cb_1_C_12_Datatype = 6
  Cb_1_C_13
  Cb_1_C_13_Name = readCoaterBk1_13
  Cb_1_C_13_Datatype = 6
  Cb_1_C_14
  Cb_1_C_14_Name = readCoaterBk1_14
  Cb_1_C_14_Datatype = 6
  Cb_1_C_15
  Cb_1_C_15_Name = readCoaterBk1_15
  Cb_1_C_15_Datatype = 6
  Cb_1_C_16
  Cb_1_C_16_Name = readCoaterBk1_16
  Cb_1_C_16_Datatype = 6
  Cb_1_C_17
  Cb_1_C_17_Name = readCoaterBk1_17
  Cb_1_C_17_Datatype = 6
  Cb_1_C_18
  Cb_1_C_18_Name = readCoaterBk1_18
  Cb_1_C_18_Datatype = 6
  Cb_1_C_19
  Cb_1_C_19_Name = readCoaterBk1_19
  Cb_1_C_19_Datatype = 6
  Cb_1_C_20
  Cb_1_C_20_Name = readCoaterBk1_20
  Cb_1_C_20_Datatype = 6
  Cb_1_C_21
  Cb_1_C_21_Name = readCoaterBk1_21
  Cb_1_C_21_Datatype = 6
  Cb_1_C_22
  Cb_1_C_22_Name = readCoaterBk1_22
  Cb_1_C_22_Datatype = 6
  Cb_1_C_23
  Cb_1_C_23_Name = readCoaterBk1_23
  Cb_1_C_23_Datatype = 6
  Cb_1_C_24
  Cb_1_C_24_Name = readCoaterBk1_24
  Cb_1_C_24_Datatype = 6
  Cb_1_C_25
  Cb_1_C_25_Name = readCoaterBk1_25
  Cb_1_C_25_Datatype = 6
  Cb_2
  Cb_2_FunCode = 16
  Cb_2_NumItemsExt = 25
  Cb_2_C_1
  Cb_2_C_1_Name = writeCoaterBk2_1
  Cb_2_C_1_Datatype = 6
  Cb_2_C_1_Dir = 1
  Cb_2_C_2
  Cb_2_C_2_Name = writeCoaterBk2_2
  Cb_2_C_2_Datatype = 6
  Cb_2_C_2_Dir = 1
  Cb_2_C_3
  Cb_2_C_3_Name = writeCoaterBk2_3
  Cb_2_C_3_Datatype = 6
  Cb_2_C_3_Dir = 1
  Cb_2_C_4
  Cb_2_C_4_Name = writeCoaterBk2_4
  Cb_2_C_4_Datatype = 6
  Cb_2_C_4_Dir = 1
  Cb_2_C_5
  Cb_2_C_5_Name = writeCoaterBk2_5
  Cb_2_C_5_Datatype = 6
  Cb_2_C_5_Dir = 1
  Cb_2_C_6
  Cb_2_C_6_Name = writeCoaterBk2_6
  Cb_2_C_6_Datatype = 6
  Cb_2_C_6_Dir = 1
  Cb_2_C_7
  Cb_2_C_7_Name = writeCoaterBk2_7
  Cb_2_C_7_Datatype = 6
  Cb_2_C_7_Dir = 1
  Cb_2_C_8
  Cb_2_C_8_Name = writeCoaterBk2_8
  Cb_2_C_8_Datatype = 6
  Cb_2_C_8_Dir = 1
  Cb_2_C_9
  Cb_2_C_9_Name = writeCoaterBk2_9
  Cb_2_C_9_Datatype = 6
  Cb_2_C_9_Dir = 1
  Cb_2_C_10
  Cb_2_C_10_Name = writeCoaterBk2_10
  Cb_2_C_10_Datatype = 6
  Cb_2_C_10_Dir = 1
  Cb_2_C_11
  Cb_2_C_11_Name = writeCoaterBk2_11
  Cb_2_C_11_Datatype = 6
  Cb_2_C_11_Dir = 1
  Cb_2_C_12
  Cb_2_C_12_Name = writeCoaterBk2_12
  Cb_2_C_12_Datatype = 6
  Cb_2_C_12_Dir = 1
  Cb_2_C_13
  Cb_2_C_13_Name = writeCoaterBk2_13
  Cb_2_C_13_Datatype = 6
  Cb_2_C_13_Dir = 1
  Cb_2_C_14
  Cb_2_C_14_Name = writeCoaterBk2_14
  Cb_2_C_14_Datatype = 6
  Cb_2_C_14_Dir = 1
  Cb_2_C_15
  Cb_2_C_15_Name = writeCoaterBk2_15
  Cb_2_C_15_Datatype = 6
  Cb_2_C_15_Dir = 1
  Cb_2_C_16
  Cb_2_C_16_Name = writeCoaterBk2_16
  Cb_2_C_16_Datatype = 6
  Cb_2_C_16_Dir = 1
  Cb_2_C_17
  Cb_2_C_17_Name = writeCoaterBk2_17
  Cb_2_C_17_Datatype = 6
  Cb_2_C_17_Dir = 1
  Cb_2_C_18
  Cb_2_C_18_Name = writeCoaterBk2_18
  Cb_2_C_18_Datatype = 6
  Cb_2_C_18_Dir = 1
  Cb_2_C_19
  Cb_2_C_19_Name = writeCoaterBk2_19
  Cb_2_C_19_Datatype = 6
  Cb_2_C_19_Dir = 1
  Cb_2_C_20
  Cb_2_C_20_Name = writeCoaterBk2_20
  Cb_2_C_20_Datatype = 6
  Cb_2_C_20_Dir = 1
  Cb_2_C_21
  Cb_2_C_21_Name = writeCoaterBk2_21
  Cb_2_C_21_Datatype = 6
  Cb_2_C_21_Dir = 1
  Cb_2_C_22
  Cb_2_C_22_Name = writeCoaterBk2_22
  Cb_2_C_22_Datatype = 6
  Cb_2_C_22_Dir = 1
  Cb_2_C_23
  Cb_2_C_23_Name = writeCoaterBk2_23
  Cb_2_C_23_Datatype = 6
  Cb_2_C_23_Dir = 1
  Cb_2_C_24
  Cb_2_C_24_Name = writeCoaterBk2_24
  Cb_2_C_24_Datatype = 6
  Cb_2_C_24_Dir = 1
  Cb_2_C_25
  Cb_2_C_25_Name = writeCoaterBk2_25
  Cb_2_C_25_Datatype = 6
  Cb_2_C_25_Dir = 1
ModbusSafety : ModbusTcp_any v1.1.0.0 (Disabled=true)  [ETH1 -> ModbusStacker.ETH2 [Cable Type=PowerlinkCable, Length=10, Version=1.0.0.3]; ETH2 -> ModbusPowerMeter.ETH1 [Cable Type=PowerlinkCable, Length=10, Version=1.0.0.3]]
  Connector ETH2 (Disabled=true)
  IpAddress = 192.168.125.50
  UnitId = 1
  Cb_1
  Cb_1_FunCode = 3
  Cb_1_Addr = 30001
  Cb_1_NumItems = 12
  Cb_1_C_1
  Cb_1_C_1_Name = readSafetyBk1_1
  Cb_1_C_1_Datatype = 6
  Cb_1_C_2
  Cb_1_C_2_Name = readSafetyBk1_2
  Cb_1_C_2_Datatype = 6
  Cb_1_C_3
  Cb_1_C_3_Name = readSafetyBk1_3
  Cb_1_C_3_Datatype = 6
  Cb_1_C_4
  Cb_1_C_4_Name = readSafetyBk1_4
  Cb_1_C_4_Datatype = 6
  Cb_1_C_5
  Cb_1_C_5_Name = readSafetyBk1_5
  Cb_1_C_5_Datatype = 6
  Cb_1_C_6
  Cb_1_C_6_Name = readSafetyBk1_6
  Cb_1_C_6_Datatype = 6
  Cb_1_C_7
  Cb_1_C_7_Name = readSafetyBk1_7
  Cb_1_C_7_Datatype = 6
  Cb_1_C_8
  Cb_1_C_8_Name = readSafetyBk1_8
  Cb_1_C_8_Datatype = 6
  Cb_1_C_9
  Cb_1_C_9_Name = readSafetyBk1_9
  Cb_1_C_9_Datatype = 6
  Cb_1_C_10
  Cb_1_C_10_Name = readSafetyBk1_10
  Cb_1_C_10_Datatype = 6
  Cb_1_C_11
  Cb_1_C_11_Name = readSafetyBk1_11
  Cb_1_C_11_Datatype = 6
  Cb_1_C_12
  Cb_1_C_12_Name = readSafetyBk1_12
  Cb_1_C_12_Datatype = 6
  Cb_2
  Cb_2_FunCode = 16
  Cb_2_AddrExt = 40001
  Cb_2_C_1
  Cb_2_C_1_Name = writeSafetyBk2_1
  Cb_2_C_1_Datatype = 6
  Cb_2_C_1_Dir = 1
ModbusStacker : ModbusTcp_any v1.1.0.0 (Disabled=true)  [ETH1 -> ModbusPrimer.ETH2 [Cable Type=PowerlinkCable, Length=10, Version=1.0.0.3]; ETH2 -> ModbusSafety.ETH1 [Cable Type=PowerlinkCable, Length=10, Version=1.0.0.3]]
  Connector ETH2 (Disabled=true)
  IpAddress = 192.168.125.185
  UnitId = 1
  Cb_1
  Cb_1_FunCode = 4
  Cb_1_NumItems = 25
  Cb_1_C_1
  Cb_1_C_1_Name = readStackerBk1_1
  Cb_1_C_1_Datatype = 6
  Cb_1_C_2
  Cb_1_C_2_Name = readStackerBk1_2
  Cb_1_C_2_Datatype = 6
  Cb_1_C_3
  Cb_1_C_3_Name = readStackerBk1_3
  Cb_1_C_3_Datatype = 6
  Cb_1_C_4
  Cb_1_C_4_Name = readStackerBk1_4
  Cb_1_C_4_Datatype = 6
  Cb_1_C_5
  Cb_1_C_5_Name = readStackerBk1_5
  Cb_1_C_5_Datatype = 6
  Cb_1_C_6
  Cb_1_C_6_Name = readStackerBk1_6
  Cb_1_C_6_Datatype = 6
  Cb_1_C_7
  Cb_1_C_7_Name = readStackerBk1_7
  Cb_1_C_7_Datatype = 6
  Cb_1_C_8
  Cb_1_C_8_Name = readStackerBk1_8
  Cb_1_C_8_Datatype = 6
  Cb_1_C_9
  Cb_1_C_9_Name = readStackerBk1_9
  Cb_1_C_9_Datatype = 6
  Cb_1_C_10
  Cb_1_C_10_Name = readStackerBk1_10
  Cb_1_C_10_Datatype = 6
  Cb_1_C_11
  Cb_1_C_11_Name = readStackerBk1_11
  Cb_1_C_11_Datatype = 6
  Cb_1_C_12
  Cb_1_C_12_Name = readStackerBk1_12
  Cb_1_C_12_Datatype = 6
  Cb_1_C_13
  Cb_1_C_13_Name = readStackerBk1_13
  Cb_1_C_13_Datatype = 6
  Cb_1_C_14
  Cb_1_C_14_Name = readStackerBk1_14
  Cb_1_C_14_Datatype = 6
  Cb_1_C_15
  Cb_1_C_15_Name = readStackerBk1_15
  Cb_1_C_15_Datatype = 6
  Cb_1_C_16
  Cb_1_C_16_Name = readStackerBk1_16
  Cb_1_C_16_Datatype = 6
  Cb_1_C_17
  Cb_1_C_17_Name = readStackerBk1_17
  Cb_1_C_17_Datatype = 6
  Cb_1_C_18
  Cb_1_C_18_Name = readStackerBk1_18
  Cb_1_C_18_Datatype = 6
  Cb_1_C_19
  Cb_1_C_19_Name = readStackerBk1_19
  Cb_1_C_19_Datatype = 6
  Cb_1_C_20
  Cb_1_C_20_Name = readStackerBk1_20
  Cb_1_C_20_Datatype = 6
  Cb_1_C_21
  Cb_1_C_21_Name = readStackerBk1_21
  Cb_1_C_21_Datatype = 6
  Cb_1_C_22
  Cb_1_C_22_Name = readStackerBk1_22
  Cb_1_C_22_Datatype = 6
  Cb_1_C_23
  Cb_1_C_23_Name = readStackerBk1_23
  Cb_1_C_23_Datatype = 6
  Cb_1_C_24
  Cb_1_C_24_Name = readStackerBk1_24
  Cb_1_C_24_Datatype = 6
  Cb_1_C_25
  Cb_1_C_25_Name = readStackerBk1_25
  Cb_1_C_25_Datatype = 6
  Cb_2
  Cb_2_FunCode = 16
  Cb_2_NumItemsExt = 25
  Cb_2_C_1
  Cb_2_C_1_Name = writeStackerBk2_1
  Cb_2_C_1_Datatype = 6
  Cb_2_C_1_Dir = 1
  Cb_2_C_2
  Cb_2_C_2_Name = writeStackerBk2_2
  Cb_2_C_2_Datatype = 6
  Cb_2_C_2_Dir = 1
  Cb_2_C_3
  Cb_2_C_3_Name = writeStackerBk2_3
  Cb_2_C_3_Datatype = 6
  Cb_2_C_3_Dir = 1
  Cb_2_C_4
  Cb_2_C_4_Name = writeStackerBk2_4
  Cb_2_C_4_Datatype = 6
  Cb_2_C_4_Dir = 1
  Cb_2_C_5
  Cb_2_C_5_Name = writeStackerBk2_5
  Cb_2_C_5_Datatype = 6
  Cb_2_C_5_Dir = 1
  Cb_2_C_6
  Cb_2_C_6_Name = writeStackerBk2_6
  Cb_2_C_6_Datatype = 6
  Cb_2_C_6_Dir = 1
  Cb_2_C_7
  Cb_2_C_7_Name = writeStackerBk2_7
  Cb_2_C_7_Datatype = 6
  Cb_2_C_7_Dir = 1
  Cb_2_C_8
  Cb_2_C_8_Name = writeStackerBk2_8
  Cb_2_C_8_Datatype = 6
  Cb_2_C_8_Dir = 1
  Cb_2_C_9
  Cb_2_C_9_Name = writeStackerBk2_9
  Cb_2_C_9_Datatype = 6
  Cb_2_C_9_Dir = 1
  Cb_2_C_10
  Cb_2_C_10_Name = writeStackerBk2_10
  Cb_2_C_10_Datatype = 6
  Cb_2_C_10_Dir = 1
  Cb_2_C_11
  Cb_2_C_11_Name = writeStackerBk2_11
  Cb_2_C_11_Datatype = 6
  Cb_2_C_11_Dir = 1
  Cb_2_C_12
  Cb_2_C_12_Name = writeStackerBk2_12
  Cb_2_C_12_Datatype = 6
  Cb_2_C_12_Dir = 1
  Cb_2_C_13
  Cb_2_C_13_Name = writeStackerBk2_13
  Cb_2_C_13_Datatype = 6
  Cb_2_C_13_Dir = 1
  Cb_2_C_14
  Cb_2_C_14_Name = writeStackerBk2_14
  Cb_2_C_14_Datatype = 6
  Cb_2_C_14_Dir = 1
  Cb_2_C_15
  Cb_2_C_15_Name = writeStackerBk2_15
  Cb_2_C_15_Datatype = 6
  Cb_2_C_15_Dir = 1
  Cb_2_C_16
  Cb_2_C_16_Name = writeStackerBk2_16
  Cb_2_C_16_Datatype = 6
  Cb_2_C_16_Dir = 1
  Cb_2_C_17
  Cb_2_C_17_Name = writeStackerBk2_17
  Cb_2_C_17_Datatype = 6
  Cb_2_C_17_Dir = 1
  Cb_2_C_18
  Cb_2_C_18_Name = writeStackerBk2_18
  Cb_2_C_18_Datatype = 6
  Cb_2_C_18_Dir = 1
  Cb_2_C_19
  Cb_2_C_19_Name = writeStackerBk2_19
  Cb_2_C_19_Datatype = 6
  Cb_2_C_19_Dir = 1
  Cb_2_C_20
  Cb_2_C_20_Name = writeStackerBk2_20
  Cb_2_C_20_Datatype = 6
  Cb_2_C_20_Dir = 1
  Cb_2_C_21
  Cb_2_C_21_Name = writeStackerBk2_21
  Cb_2_C_21_Datatype = 6
  Cb_2_C_21_Dir = 1
  Cb_2_C_22
  Cb_2_C_22_Name = writeStackerBk2_22
  Cb_2_C_22_Datatype = 6
  Cb_2_C_22_Dir = 1
  Cb_2_C_23
  Cb_2_C_23_Name = writeStackerBk2_23
  Cb_2_C_23_Datatype = 6
  Cb_2_C_23_Dir = 1
  Cb_2_C_24
  Cb_2_C_24_Name = writeStackerBk2_24
  Cb_2_C_24_Datatype = 6
  Cb_2_C_24_Dir = 1
  Cb_2_C_25
  Cb_2_C_25_Name = writeStackerBk2_25
  Cb_2_C_25_Datatype = 6
  Cb_2_C_25_Dir = 1
OpcUaDryer : OpcUa_any v1.0.0.1 (Disabled=true)  [ETH1 -> ModbusPowerMeter.ETH2 [Cable Type=PowerlinkCable, Length=10, Version=1.0.0.3]]
  Connector ETH2 (Disabled=true)
  ServerEndpointUrl = opc.tcp://192.168.125.47:4840
  UserIdentifyToken = 1
  Username = Printer_user
  Password = h98o76
  Channel1
  ChannelID1 = xError
  ChannelBrowsePath1 = /0:Root/0:Objects/4:PLC/6:Modules/6:&:&:/6:Global PV/6:gDryerLocalData/6:xError
  Channel2
  ChannelID2 = xDrying
  ChannelBrowsePath2 = /0:Root/0:Objects/4:PLC/6:Modules/6:&:&:/6:Global PV/6:gDryerLocalData/6:xDrying
  Channel3
  ChannelID3 = xReadyToDry
  ChannelBrowsePath3 = /0:Root/0:Objects/4:PLC/6:Modules/6:&:&:/6:Global PV/6:gDryerLocalData/6:xReadyToDry
  Channel4
  ChannelID4 = xJamDetection
  ChannelBrowsePath4 = /0:Root/0:Objects/4:PLC/6:Modules/6:&:&:/6:Global PV/6:gDryerLocalData/6:xJamDetection
  Channel5
  ChannelID5 = xTransportMoving
  ChannelBrowsePath5 = /0:Root/0:Objects/4:PLC/6:Modules/6:&:&:/6:Global PV/6:gDryerLocalData/6:xTransportMoving
  Channel6
  ChannelID6 = xInRemote
  ChannelBrowsePath6 = /0:Root/0:Objects/4:PLC/6:Modules/6:&:&:/6:Global PV/6:gDryerLocalData/6:xInRemote
PC_any : PC_any v1.1.1.0 (OrderNumber=PC)
  Connector IF3:
    ActivateIna = 0
    Vnc1
    VncVcObjectName1 = SimVis
    VncKeyMappingFile1 = VC\PS2-Keyboard.dis
    VncPortNumber1 = 5901
    VncMaxConnections1 = 4
    VncRefreshRate1 = 250
    VncTitle1 = EFI_printer_Sim
    Vnc2
    VncKeyMappingFile2 = VC\PS2-Keyboard1.dis
    VncMaxConnections2 = 4
    VncRefreshRate2 = 250
    VncTitle2 = EFI_printer_Inks
    Vnc3
    VncVcObjectName3 = Panel
    VncKeyMappingFile3 = VC\PS2-Keyboard2.dis
    VncPortNumber3 = 5903
    VncMaxConnections3 = 2
    VncRefreshRate3 = 500
    VncTitle3 = EFI_Safety_Transfer
    Vnc4
    VncKeyMappingFile4 = VC\PS2-Keyboard3.dis
    VncPortNumber4 = 5902
    VncRefreshRate4 = 300
    VncTitle4 = Diagnostic Screen
  ConfigurationID = SimTests
  PermanentPvSize = 24000
  RemanentGlobalPvSize = 10000
  VolatileGlobalPvSize = 1600000
  SystemTick = 2000
  Cyclic1Duration = 4000
  Cyclic1Tolerance = 0
  Cyclic1Stack = 32768
  Cyclic2Duration = 8000
  Cyclic2Tolerance = 0
  Cyclic2Stack = 32768
  Cyclic3Duration = 16000
  Cyclic3Tolerance = 16000
  Cyclic3Stack = 32768
  Cyclic4Duration = 32000
  Cyclic4Tolerance = 32000
  Cyclic4Stack = 32768
  Cyclic5Duration = 80000
  Cyclic5Tolerance = 80000
  Cyclic5Stack = 32768
  Cyclic6Duration = 88000
  Cyclic6Tolerance = 88000
  Cyclic6Stack = 32768
  Cyclic7Duration = 44000
  Cyclic7Tolerance = 88000
  Cyclic7Stack = 32768
  Cyclic8Duration = 16000
  Cyclic8Tolerance = 16000
  Cyclic8Stack = 32768
  FileDevice1
  FileDeviceName1 = USER
  FileDevicePath1 = USER_PATH
  FtpUser1
  FtpUsername1 = P4  // P4
  FtpUserPassword1 = LclxNYuP61nqo0LTZcDXp7yBDKZw4k3sO5UoQKFs6g8=  // efi
  FtpUserSalt1 = Ni00Nvek
  FTPAccessRight1 = 0
  WebServerPort = 82
  ActivateOpcUa = 1
  OpcUa_Limits_MonitoredItemsPerSubscription = 2500
  OpcUaMaxSubsEventQueueSize = 2500
  OpcUa_Limits_MinPublishingIntervall = 100
  OpcUa_Limits_MinKeepAlive = 200
  OpcUaInformationModels_PV_Version = 2
  OpcUaInformationModel_Facet = 0
  OpcUaInformationModel_TypeInformation = 0
  OpcUaInformationModel_BaseObjectTypeForStructures = 0
X67SM2436 : X67SM2436 v2.3.0.0  [X2X1 -> 5LS197.6.IF2 [Cable Type=X2XCable, Length=10, Version=1.0.0.3]]
```

### Cpu.per - PC_any/Cpu.per
```iecst
VAR_CONFIG
	gPermanentSN AT %M0; (*Serial Number of the machine*)
	gPermanentVersion AT %M100; (* *)
	gPermanentSimMachinePar AT %M116; (* *)
	gPermanentMachine AT %M150; (* *)
	gPermanentBlock AT %M1300; (* *)
	gPermanentAnalogSensor AT %M1500; (* *)
	gInksPermanentParBar AT %M2700; (* *)
	HoldingRegister AT %MW6000; (* *)
END_VAR
```
